// TwinCAT 3 PLC project mover_demo
// ProgramVersion: 3.1.4024.12
// libraries:
//   CmpBitmapPool, * (System)
//   Tc2_Math, * (Beckhoff Automation GmbH)
//   Tc2_MC2, * (Beckhoff Automation GmbH)
//   Tc2_MC2_Drive, * (Beckhoff Automation GmbH)
//   Tc2_Standard, * (Beckhoff Automation GmbH)
//   Tc2_System, * (Beckhoff Automation GmbH)
//   Tc2_Utilities, * (Beckhoff Automation GmbH)
//   Tc3_JsonXml, * (Beckhoff Automation GmbH)
//   Tc3_Module, * (Beckhoff Automation GmbH)
//   VisuDialogs, * (System)
//   VisuSymbols,3.5.10.0,System
// project tree:
//   DUTs/Helptec/Axis/ AxisBase_t.TcDUT, AxisBeckhoff_t.TcDUT, AxisLinMotConst_t.TcDUT (not stored), AxisLinMot_t.TcDUT, AxisSMC_t.TcDUT (not stored), typeInputArea.TcDUT, typeOutputArea.TcDUT
//   DUTs/Helptec/ Cylinder2Pos_config.TcDUT, enLamp.TcDUT (not stored), enState.TcDUT (not stored), structAlarm.TcDUT (not stored), structButton.TcDUT
//   DUTs/Helptec/Recipe/ RecipeAxisLinear2Pos_t.TcDUT
//   DUTs/Helptec/RS_Axis/ FeederDelays_t.TcDUT (not stored), MoveProfile1D_t.TcDUT, MoveProfile_t.TcDUT, TriggerType_e.TcDUT, VectorMove1D_t.TcDUT
//   DUTs/ PieceType_e.TcTLEO (not stored), Mover_st.TcDUT (not stored), Piece_st.TcDUT (not stored)
//   / GlobalTextList.TcGTLO (excluded from build), PlcTask.TcTTO, Visualization Manager.TcVMO (not stored), VISU_TASK.TcTTO
//   GVLs/ AXIS.TcGVL, CONST.TcGVL, GVL.TcGVL, HMI.TcGVL, IN.TcGVL, IO_BOX.TcGVL, OUT.TcGVL, PERS.TcGVL, SIMU.TcGVL
//   POUs/00_MAIN/FB%27s/ FB_Safety.TcPOU (not stored)
//   POUs/00_MAIN/ MAIN.TcPOU, _02_SAFETY.TcPOU, _05_FLAGS.TcPOU (not stored)
//   POUs/10_HMI/FB%27s/ FB_BUTTON.TcPOU (not stored), FB_HMI_BT.TcPOU (not stored), FB_Keba_key.TcPOU (not stored), FB_LampeBNI007F.TcPOU (not stored), FB_STATE.TcPOU (not stored)
//   POUs/10_HMI/ _10_HMI.TcPOU, _11_PAR_CHK.TcPOU (not stored), _14_STATE.TcPOU
//   POUs/20_AUTO/ Axis_e.TcTLEO, LinearAxis_e.TcTLEO, RecipeType_e.TcTLEO, Recipe_21_101_t.TcDUT, StationList_e.TcTLEO, _20_AUTO.TcPOU, _21_CopyDefaultRecipe.TcPOU
//   POUs/20_AUTO/BuR SuperTrack com/ CT_Shuttle_BR_to_Tc_Status_t.TcDUT, CT_Shuttle_BR_to_Tc_t.TcDUT, CT_Shuttle_BR_to_Tc_u.TcDUT, CT_Shuttle_Tc_To_BR_Command_t.TcDUT, CT_Shuttle_Tc_to_BR_t.TcDUT, CT_Shuttle_Tc_to_BR_u.TcDUT, CT_Track_BR_to_TC_Status_t.TcDUT, CT_Track_BR_to_Tc_t.TcDUT, CT_Track_BR_to_Tc_u.TcDUT, CT_Track_Tc_to_BR_Command_t.TcDUT, CT_Track_Tc_to_BR_t.TcDUT, CT_Track_Tc_to_BR_u.TcDUT, gMoverAxis.TcGVL
//   POUs/20_AUTO/FB%27s/Alarm/ FB_ALARM.TcPOU (not stored), FB_ALARM32.TcPOU (not stored)
//   POUs/20_AUTO/FB%27s/ FB_WandlerForceSensor.TcPOU (not stored), getPercent.TcPOU (not stored)
//   POUs/20_AUTO/FB%27s/RS Axis/ BowlBandFeeder_Config_t.TcDUT (not stored), FB_AUT_Statistics.TcPOU (not stored), FB_BowlBandFeeder.TcPOU (not stored), FB_Feeder2Sensors.TcPOU (not stored), FB_Fifo.TcPOU (not stored), FB_LinearMotionMan.TcPOU (not stored), LinearMotionMan_Config_t.TcDUT (not stored)
//   POUs/20_AUTO/FB%27s/Achsen/ FB_AxisLIN_V1_1.TcPOU (not stored), FB_AxisLMturn_V1_1.TcPOU (not stored), FB_AxisLM_V1_1.TcPOU (not stored), FB_AxisRotTable_V1_1.TcPOU (not stored), FB_AxisSMC_V1_1.TcPOU (not stored), FB_AxisTURN_V1_1.TcPOU (not stored), JXCE1_Baustein.TcPOU (not stored)
//   POUs/20_AUTO/FB%27s/Pneumatic/ FB_ZylMo2El_V2_1.TcPOU (not stored)
//   POUs/20_AUTO/FB%27s/Vorlagen/ FB_ABL_VORLAGE.TcPOU (not stored), POU_AUT_VORLAGE.TcPOU (not stored), POU_ERR_VORLAGE.TcPOU (not stored), _01_MAIN.TcPOU (not stored)
//   POUs/20_AUTO/FileMan/ FB_FileMan.TcPOU, FileMan.TcPOU, LoadFromMemory.TcPOU, ReadJsonDom.TcPOU, SaveInMemory.TcPOU, SaveInMemory_Recipe.TcPOU
//   POUs/20_AUTO/Mover/ ApproachScenario_e.TcTLEO, DistToTravel.TcPOU, FB_Group.TcPOU, FB_Mover.TcPOU, FB_MoverMan.TcPOU, FB_Position.TcPOU, FB_SimuMoverAxis.TcPOU, FB_Station.TcPOU, FB_PieceHolder.TcPOU, FB_StationMan.TcPOU, IProcessSampleMover.TcIO (not stored), ISimuMoverTimers.TcIO, IStation.TcIO, MoverDirection_e.TcTLEO, MoverState_e.TcTLEO, VISU_MoverDetail.TcVIS, VISU_MoverView.TcVIS, Pos2D_t.TcDUT (not stored), ProcessExec_e.TcDUT (not stored), StationName_e.TcTLEO
//   POUs/20_AUTO/Simu/ FB_Simu_AxisLIN_V1_1.TcPOU, FB_Simu_AxisLM_V1_1.TcPOU, FB_Simu_Feeder.TcPOU, FB_Simu_Zyl2Pos.TcPOU
//   POUs/20_AUTO/ST100/ FB_ABL_LASER.TcPOU, FB_AUT_LASER.TcPOU, FB_AUT_100.TcPOU, F_GetPercent.TcPOU (not stored), F_GetPercent_2.TcPOU, ST100_Load_e.TcTLEO (not stored), FB_ABL_LOAD.TcPOU, FB_ABL_MODIFY.TcPOU, FB_ABL_UNLOAD.TcPOU, FB_AUT_ABSTRACT.TcPOU, FB_ABL_100.TcPOU (not stored), FB_AUT_LOAD.TcPOU, FB_AUT_MODIFY.TcPOU, FB_AUT_UNLOAD.TcPOU, ProcessExecution_e.TcTLEO (not stored), ST100_e.TcTLEO (not stored), ST100_Modify_e.TcTLEO (not stored), ST100_Laser_e.TcTLEO, ST100_Unload_e.TcTLEO (not stored)
//   POUs/20_AUTO/ST105/Fanuc_robot/ Fanuc_command_ext_to_robot_t.TcDUT (not stored), Fanuc_command_std_to_robot_t.TcDUT, Fanuc_hw_command_to_robot_t.TcDUT (not stored), Fanuc_status_std_from_robot.TcDUT (not stored), ST105_Fanuc_command_t.TcDUT, ST105_Fanuc_status_t.TcDUT
//   POUs/20_AUTO/ST105/ FB_ABL_105_Feeder.TcPOU, FB_ABL_105_Pnp.TcPOU, FB_AUT_105.TcPOU, ST105_Axis.TcGVL, ST105_PnpVerPushPos_e.TcDUT, ST105_Recipe_t.TcDUT, ST105_Feeder_e.TcDUT, ST105_Pnp_e.TcTLEO, ST105_Slider_e.TcDUT, ST105_Cylinders_e.TcTLEO, VISU_Recipe_ST105.TcVIS, VISU_ST105.TcVIS
//   POUs/20_AUTO/ST110/ POU_ALARM_110.TcPOU, ST110_Alarm_e.TcDUT, ST110_Cylinders_e.TcTLEO (not stored), ST110_Feeder_e.TcDUT, FB_ABL_110_Feeder.TcPOU, FB_ABL_110_Pnp.TcPOU, FB_AUT_110.TcPOU, ST110_Axis.TcGVL, ST110_PnpVerPushPos_e.TcDUT, ST110_Pnp_e.TcTLEO, ST110_PnpHorPos_e.TcDUT, ST110_PnpVerPos_e.TcDUT, ST110_Recipe_t.TcDUT, VISU_Recipe_ST110.TcVIS, VISU_ST110.TcVIS
//   POUs/20_AUTO/ST115/ FB_ABL_115_Feeder.TcPOU, FB_ABL_115_Pnp.TcPOU, FB_AUT_115.TcPOU, ST115_PnpVerPushPos_e.TcDUT, ST115_Cylinders_e.TcTLEO, ST115_Recipe_t.TcDUT, ST115_Axis.TcGVL, ST115_Feeder_e.TcDUT, ST115_PnpHorPos_e.TcDUT, ST115_PnpVerPos_e.TcDUT (not stored), ST115_Pnp_e.TcTLEO, VISU_Recipe_ST115.TcVIS, VISU_ST115.TcVIS
//   POUs/20_AUTO/ST120/ FB_ABL_120_Feeder.TcPOU, FB_ABL_120_Pnp.TcPOU, FB_AUT_120.TcPOU, POU_ALARM_120.TcPOU (not stored), ST120_Alarm_e.TcDUT (not stored), ST120_Cylinders_e.TcTLEO, ST120_Axis.TcGVL, ST120_Feeder_e.TcDUT, ST120_PnpHorPos_e.TcDUT (not stored), ST120_PnpVerPos_e.TcDUT, ST120_Pnp_e.TcTLEO, ST120_Recipe_t.TcDUT, VISU_Recipe_ST120.TcVIS, VISU_ST120.TcVIS
//   POUs/20_AUTO/ST125/ FB_ABL_125_Feeder.TcPOU, FB_ABL_125_Pnp.TcPOU, FB_AUT_125.TcPOU, POU_ALARM_125.TcPOU, ST125_Alarm_e.TcDUT, ST125_Cylinders_e.TcTLEO, ST125_Axis.TcGVL, ST125_Feeder_e.TcDUT, ST125_PnpHorPos_e.TcDUT, ST125_PnpVerPos_e.TcDUT, ST125_Pnp_e.TcTLEO, ST125_Recipe_t.TcDUT, VISU_Recipe_ST125.TcVIS, VISU_ST125.TcVIS
//   POUs/20_AUTO/ST128/ FB_ABL_128_TubeCapCheck.TcPOU, FB_AUT_128.TcPOU, ST128_TubeCapCheck_e.TcTLEO (not stored), ST128_Recipe_t.TcDUT, VISU_Recipe_ST128.TcVIS (not stored), VISU_ST128.TcVIS
//   POUs/20_AUTO/ST130/ FB_ABL_130_Dose.TcPOU, FB_ABL_MODIFY_135.TcPOU, FB_AUT_130.TcPOU, FB_AUT_135.TcPOU, ST130_Axis.TcGVL, ST130_Cylinders_e.TcTLEO, ST130_DosierkammerPos_e.TcDUT (not stored), ST130_PatroneAushebenPos_e.TcDUT, ST130_Recipe_t.TcDUT, ST130_Dose_e.TcTLEO, VISU_Recipe_ST130.TcVIS, VISU_ST130.TcVIS
//   POUs/20_AUTO/ST140/ FB_ABL_140_Measure.TcPOU, FB_AUT_140.TcPOU, LaserPlace_e.TcDUT, ST140_Measure_e.TcTLEO, ST140_Recipe_t.TcDUT, VISU_Recipe_ST140.TcVIS, VISU_ST140.TcVIS
//   POUs/20_AUTO/ST145/ FB_ABL_145_Feeder.TcPOU, FB_ABL_145_Pnp.TcPOU, FB_AUT_145.TcPOU, ST145_Axis.TcGVL, ST145_Cylinders_e.TcTLEO (not stored), ST145_Feeder_e.TcDUT, ST145_PnpHorPos_e.TcDUT, ST145_PnpVerPos_e.TcDUT, ST145_Recipe_t.TcDUT, ST145_Pnp_e.TcTLEO, VISU_Recipe_ST145.TcVIS, VISU_ST145.TcVIS
//   POUs/20_AUTO/ST15x/ FB_ABL_150.TcPOU, FB_ABL_150_solo.TcPOU, FB_AUT_150.TcPOU, FB_AUT_155.TcPOU, ST150_Cylinders_e.TcTLEO, ST150_Uss_e.TcTLEO, ST150_Recipe_t.TcDUT (not stored), Ultrasonic_IN_bits_t.TcDUT, Ultrasonic_OUT_bits_t.TcDUT, VISU_Recipe_ST150.TcVIS, VISU_ST150.TcVIS
//   POUs/20_AUTO/ST16x/CETA/ CETA_error_handling_t.TcDUT, CETA_IN_bits_t.TcDUT, CETA_IN_u.TcDUT, CETA_IO.TcGVL, CETA_OUT_bits_t.TcDUT, CETA_OUT_u.TcDUT, CETA_Result_e.TcDUT, CETA_Unit_e.TcDUT, FB_CETA_715.TcPOU
//   POUs/20_AUTO/ST16x/CETA/CETA_Measurement_t/ CETA_Measurement_block1_t.TcDUT (not stored), CETA_Measurement_block2_t.TcDUT, CETA_Measurement_block3_t.TcDUT (not stored), CETA_Measurement_t.TcDUT, CETA_Res_Data_t.TcDUT
//   POUs/20_AUTO/ST16x/CETA/CETA_Parameter_blocks/ CETA_Parameter_blocks_t.TcDUT
//   POUs/20_AUTO/ST16x/CETA/CETA_com_union/ CETA_Parameter_blocks_u.TcDUT
//   POUs/20_AUTO/ST16x/ FB_ABL_160.TcPOU, FB_AUT_160.TcPOU, FB_AUT_165.TcPOU, ST160_PnpVerPos_e.TcDUT, ST16x_Axis.TcGVL, ST160_Cylinders_e.TcTLEO, ST160_Recipe_t.TcDUT, ST160_CETA_e.TcTLEO, VISU_Recipe_ST160.TcVIS, VISU_ST160.TcVIS
//   POUs/20_AUTO/ST170/ FB_ABL_170.TcPOU, FB_AUT_170.TcPOU, ST170_Axis.TcGVL (not stored), ST170_RFID_e.TcTLEO, ST170_PnpVerPos_e.TcDUT, ST170_Recipe_t.TcDUT, VISU_Recipe_ST170.TcVIS, VISU_ST170.TcVIS
//   POUs/20_AUTO/ST175/ FB_ABL_175.TcPOU, FB_AUT_175.TcPOU, ST175_LASER_e.TcTLEO, ST175_Cylinders_e.TcTLEO, ST175_Recipe_t.TcDUT, VISU_Recipe_ST175.TcVIS, VISU_ST175.TcVIS (not stored)
//   POUs/20_AUTO/ST175/Trumpf/ FB_Laser_ABL.TcPOU, if_BitCommand_u.TcDUT (not stored), if_Command_t.TcDUT, if_Command_u.TcDUT, if_SingleCmds.TcGVL (not stored), if_TruMark.TcGVL, TruMarkLaserStatus.TcDUT (not stored), TruMark_Ethercat_dj.TcPOU, TruMark_SingleCmds.TcPOU
//   POUs/20_AUTO/ST180/ FB_ABL_180_Pnp.TcPOU, FB_AUT_180.TcPOU, ST180_Axis.TcGVL, ST180_Cylinders_e.TcTLEO, ST180_PnpHorPos_e.TcDUT (not stored), ST180_PnpVerPos_e.TcDUT, ST180_Pnp_e.TcTLEO, ST180_Recipe_t.TcDUT, VISU_Recipe_ST180.TcVIS, VISU_ST180.TcVIS
//   POUs/20_AUTO/ST185/ FB_ABL_185_Pnp.TcPOU, FB_AUT_185.TcPOU, ST185_Axis.TcGVL, ST185_Cylinders_e.TcTLEO, ST185_PnpHorPos_e.TcDUT, ST185_PnpVerPos_e.TcDUT, ST185_Pnp_e.TcTLEO, ST185_Recipe_t.TcDUT, VISU_Recipe_ST185.TcVIS, VISU_ST185.TcVIS (not stored)
//   POUs/20_AUTO/TOOL/ ASSERT.TcPOU, EqualApproximately.TcPOU (not stored), EqualDelta.TcPOU (not stored), EqualEssentially.TcPOU (not stored), GetTick.TcPOU, IObject.TcIO, MAP_REAL_TO_INT.TcPOU, SortBubbleLREAL.TcPOU (not stored)
//   VISUs/ Custom.TcIPO (not stored), VISU_LinearConfigArray.TcVIS, VISU_Cylinder2PosConfig.TcVIS, VISU_AxisManual.TcVIS, VISU_main.TcVIS, VISU_Time.TcVIS
// real-time tasks:
//   TASK PlcTask: cycle T#10ms, priority 20, ADS port 350
//   TASK VISU_TASK: cycle T#10ms, priority 21, ADS port 351
//   TASK Task_fileMan: cycle T#100000us, priority 45, ADS port 352
// motion (NC):
//   TASK NC-Task 1 SAF: cycle T#2ms, priority 4, ADS port 501
//   TASK NC-Task 1 SVB: cycle T#10ms, priority 8, ADS port 511
//   AXIS ST110_01Y (id 1)
//     Dynamic: AccelerationMaximum=100000, DecelerationMaximum=100000, Acceleration=40000, Deceleration=40000, Jerk=800000
//     OtherSettings: AllowMotionCmdToSlave=true
//     encoder EncType=1
//       SoftEndMinControl: Enable=true, Range=-5
//     drive DrvType=5
//       Analog: TorqueSetpointScale=10, ScaleFactorActTorque=0.1
//       TimeComp: TaskDelayCycles=1
//     controller CtrType=1
//       CtrPara: PriorControlFactor=1
//         Observer: BandWidth=20
//   AXIS ST110_02Z (id 2)
//     Dynamic: AccelerationMaximum=100000, DecelerationMaximum=100000, Acceleration=15000, Deceleration=15000, Jerk=10000000
//     OtherSettings: AllowMotionCmdToSlave=true
//     encoder EncType=1
//       SoftEndMinControl: Enable=true, Range=-5
//     drive DrvType=5
//       Analog: TorqueSetpointScale=10, ScaleFactorActTorque=0.1
//       TimeComp: TaskDelayCycles=1
//     controller CtrType=1
//       CtrPara: PriorControlFactor=1
//         Observer: BandWidth=20
//   AXIS ST110_03Z (id 3)
//     Dynamic: AccelerationMaximum=100000, DecelerationMaximum=100000, Acceleration=15000, Deceleration=15000, Jerk=10000000
//     OtherSettings: AllowMotionCmdToSlave=true
//     encoder EncType=1
//       SoftEndMinControl: Enable=true, Range=-5
//     drive DrvType=5
//       Analog: TorqueSetpointScale=10, ScaleFactorActTorque=0.1
//       TimeComp: TaskDelayCycles=1
//     controller CtrType=1
//       CtrPara: PriorControlFactor=1
//         Observer: BandWidth=20
//   AXIS ST110_04Z (id 11)
//     OtherSettings: AllowMotionCmdToSlave=true
//     encoder EncType=1
//     drive DrvType=5
//       Analog: TorqueSetpointScale=10, ScaleFactorActTorque=0.1
//       TimeComp: TaskDelayCycles=1
//     controller CtrType=1
//       CtrPara: PriorControlFactor=1
//         Observer: BandWidth=20
//   AXIS ST110_10W (id 4)
//     General: UnitName=°, UnitFlags=#x00000004
//     Dynamic: AccelerationMaximum=36000, DecelerationMaximum=36000, Acceleration=3600, Deceleration=3600, Jerk=3600000
//     Velo: Maximum=360
//     OtherSettings: AllowMotionCmdToSlave=true
//     encoder EncType=1
//     drive DrvType=5
//       Analog: VeloReferenz=360, TorqueSetpointScale=10, ScaleFactorActTorque=0.1
//       TimeComp: TaskDelayCycles=1
//     controller CtrType=1
//       CtrPara: PriorControlFactor=1
//         Observer: BandWidth=20
//   AXIS ST115_01Y (id 5)
//     OtherSettings: AllowMotionCmdToSlave=true
//     encoder EncType=1
//     drive DrvType=5
//       Analog: TorqueSetpointScale=10, ScaleFactorActTorque=0.1
//       TimeComp: TaskDelayCycles=1
//     controller CtrType=1
//       CtrPara: PriorControlFactor=1
//         Observer: BandWidth=20
//   AXIS ST115_02Z (id 6)
//     OtherSettings: AllowMotionCmdToSlave=true
//     encoder EncType=1
//     drive DrvType=5
//       Analog: TorqueSetpointScale=10, ScaleFactorActTorque=0.1
//       TimeComp: TaskDelayCycles=1
//     controller CtrType=1
//       CtrPara: PriorControlFactor=1
//         Observer: BandWidth=20
//   AXIS ST115_03Z (id 7)
//     OtherSettings: AllowMotionCmdToSlave=true
//     encoder EncType=1
//     drive DrvType=5
//       Analog: TorqueSetpointScale=10, ScaleFactorActTorque=0.1
//       TimeComp: TaskDelayCycles=1
//     controller CtrType=1
//       CtrPara: PriorControlFactor=1
//         Observer: BandWidth=20
//   AXIS ST115_04Z (id 12)
//     OtherSettings: AllowMotionCmdToSlave=true
//     encoder EncType=1
//     drive DrvType=5
//       Analog: TorqueSetpointScale=10, ScaleFactorActTorque=0.1
//       TimeComp: TaskDelayCycles=1
//     controller CtrType=1
//       CtrPara: PriorControlFactor=1
//         Observer: BandWidth=20
//   AXIS ST115_10W (id 8)
//     General: UnitName=°
//     OtherSettings: AllowMotionCmdToSlave=true
//     encoder EncType=1
//     drive DrvType=5
//       Analog: TorqueSetpointScale=10, ScaleFactorActTorque=0.1
//       TimeComp: TaskDelayCycles=1
//     controller CtrType=1
//       CtrPara: PriorControlFactor=1
//         Observer: BandWidth=20
//   AXIS ST120_01Y (id 9)
//     OtherSettings: AllowMotionCmdToSlave=true
//     encoder EncType=1
//     drive DrvType=5
//       Analog: TorqueSetpointScale=10, ScaleFactorActTorque=0.1
//       TimeComp: TaskDelayCycles=1
//     controller CtrType=1
//       CtrPara: PriorControlFactor=1
//         Observer: BandWidth=20
//   AXIS ST120_02Z (id 10)
//     OtherSettings: AllowMotionCmdToSlave=true
//     encoder EncType=1
//     drive DrvType=5
//       Analog: TorqueSetpointScale=10, ScaleFactorActTorque=0.1
//       TimeComp: TaskDelayCycles=1
//     controller CtrType=1
//       CtrPara: PriorControlFactor=1
//         Observer: BandWidth=20
//   AXIS ST125_01Y (id 13)
//     OtherSettings: AllowMotionCmdToSlave=true
//     encoder EncType=1
//     drive DrvType=5
//       Analog: TorqueSetpointScale=10, ScaleFactorActTorque=0.1
//       TimeComp: TaskDelayCycles=1
//     controller CtrType=1
//       CtrPara: PriorControlFactor=1
//         Observer: BandWidth=20
//   AXIS ST125_02Z (id 14)
//     OtherSettings: AllowMotionCmdToSlave=true
//     encoder EncType=1
//     drive DrvType=5
//       Analog: TorqueSetpointScale=10, ScaleFactorActTorque=0.1
//       TimeComp: TaskDelayCycles=1
//     controller CtrType=1
//       CtrPara: PriorControlFactor=1
//         Observer: BandWidth=20
//   AXIS ST125_10W (id 15)
//     General: UnitName=°
//     OtherSettings: AllowMotionCmdToSlave=true
//     encoder EncType=1
//     drive DrvType=5
//       Analog: TorqueSetpointScale=10, ScaleFactorActTorque=0.1
//       TimeComp: TaskDelayCycles=1
//     controller CtrType=1
//       CtrPara: PriorControlFactor=1
//         Observer: BandWidth=20
//   AXIS SIMU_ST145_01Y (id 16)
//     OtherSettings: AllowMotionCmdToSlave=true
//     encoder EncType=1
//     drive DrvType=5
//       Analog: TorqueSetpointScale=10, ScaleFactorActTorque=0.1
//       TimeComp: TaskDelayCycles=1
//     controller CtrType=1
//       CtrPara: PriorControlFactor=1
//         Observer: BandWidth=20
//   AXIS SIMU_ST145_02Z (id 17)
//     OtherSettings: AllowMotionCmdToSlave=true
//     encoder EncType=1
//     drive DrvType=5
//       Analog: TorqueSetpointScale=10, ScaleFactorActTorque=0.1
//       TimeComp: TaskDelayCycles=1
//     controller CtrType=1
//       CtrPara: PriorControlFactor=1
//         Observer: BandWidth=20
//   AXIS ST145_10W (id 18)
//     General: UnitName=°
//     OtherSettings: AllowMotionCmdToSlave=true
//     encoder EncType=1
//     drive DrvType=5
//       Analog: TorqueSetpointScale=10, ScaleFactorActTorque=0.1
//       TimeComp: TaskDelayCycles=1
//     controller CtrType=1
//       CtrPara: PriorControlFactor=1
//         Observer: BandWidth=20
//   AXIS ST160_01Z (id 27)
//     OtherSettings: AllowMotionCmdToSlave=true
//     encoder EncType=1
//     drive DrvType=5
//       Analog: TorqueSetpointScale=10, ScaleFactorActTorque=0.1
//       TimeComp: TaskDelayCycles=1
//     controller CtrType=1
//       CtrPara: PriorControlFactor=1
//         Observer: BandWidth=20
//   AXIS ST165_01Z (id 28)
//     OtherSettings: AllowMotionCmdToSlave=true
//     encoder EncType=1
//     drive DrvType=5
//       Analog: TorqueSetpointScale=10, ScaleFactorActTorque=0.1
//       TimeComp: TaskDelayCycles=1
//     controller CtrType=1
//       CtrPara: PriorControlFactor=1
//         Observer: BandWidth=20
//   AXIS ST170_01Z (id 19)
//     OtherSettings: AllowMotionCmdToSlave=true
//     encoder EncType=1
//     drive DrvType=5
//       Analog: TorqueSetpointScale=10, ScaleFactorActTorque=0.1
//       TimeComp: TaskDelayCycles=1
//     controller CtrType=1
//       CtrPara: PriorControlFactor=1
//         Observer: BandWidth=20
//   AXIS ST180_01Y (id 20)
//     OtherSettings: AllowMotionCmdToSlave=true
//     encoder EncType=1
//     drive DrvType=5
//       Analog: TorqueSetpointScale=10, ScaleFactorActTorque=0.1
//       TimeComp: TaskDelayCycles=1
//     controller CtrType=1
//       CtrPara: PriorControlFactor=1
//         Observer: BandWidth=20
//   AXIS ST180_02Z (id 21)
//     OtherSettings: AllowMotionCmdToSlave=true
//     encoder EncType=1
//     drive DrvType=5
//       Analog: TorqueSetpointScale=10, ScaleFactorActTorque=0.1
//       TimeComp: TaskDelayCycles=1
//     controller CtrType=1
//       CtrPara: PriorControlFactor=1
//         Observer: BandWidth=20
//   AXIS ST180_10Z (id 22)
//     OtherSettings: AllowMotionCmdToSlave=true
//     encoder EncType=1
//     drive DrvType=5
//       Analog: TorqueSetpointScale=10, ScaleFactorActTorque=0.1
//       TimeComp: TaskDelayCycles=1
//     controller CtrType=1
//       CtrPara: PriorControlFactor=1
//         Observer: BandWidth=20
//   AXIS ST185_01Y (id 23)
//     OtherSettings: AllowMotionCmdToSlave=true
//     encoder EncType=1
//     drive DrvType=5
//       Analog: TorqueSetpointScale=10, ScaleFactorActTorque=0.1
//       TimeComp: TaskDelayCycles=1
//     controller CtrType=1
//       CtrPara: PriorControlFactor=1
//         Observer: BandWidth=20
//   AXIS ST185_02Z (id 24)
//     OtherSettings: AllowMotionCmdToSlave=true
//     encoder EncType=1
//     drive DrvType=5
//       Analog: TorqueSetpointScale=10, ScaleFactorActTorque=0.1
//       TimeComp: TaskDelayCycles=1
//     controller CtrType=1
//       CtrPara: PriorControlFactor=1
//         Observer: BandWidth=20
//   AXIS ST185_10Z (id 25)
//     OtherSettings: AllowMotionCmdToSlave=true
//     encoder EncType=1
//     drive DrvType=5
//       Analog: TorqueSetpointScale=10, ScaleFactorActTorque=0.1
//       TimeComp: TaskDelayCycles=1
//     controller CtrType=1
//       CtrPara: PriorControlFactor=1
//         Observer: BandWidth=20
//   AXIS Axis 34 (id 34)
//     OtherSettings: AllowMotionCmdToSlave=true
//     encoder EncType=19
//       EncPara: MaxCount=#xffffffff
//     drive DrvType=16
//       DrvPara: MaxCount=#xffffffff
//         Analog: TorqueSetpointScale=10, ScaleFactorActTorque=0.1
//         TimeComp: TaskDelayCycles=1
//     controller CtrType=1
//       CtrPara: PriorControlFactor=1
//         Observer: BandWidth=20
//   AXIS Axis 35 (id 35)
//     OtherSettings: AllowMotionCmdToSlave=true
//     encoder EncType=19
//       EncPara: MaxCount=#xffffffff
//     drive DrvType=16
//       DrvPara: MaxCount=#xffffffff
//         Analog: TorqueSetpointScale=10, ScaleFactorActTorque=0.1
//         TimeComp: TaskDelayCycles=1
//     controller CtrType=1
//       CtrPara: PriorControlFactor=1
//         Observer: BandWidth=20
//   AXIS Axis 36 (id 36)
//     OtherSettings: AllowMotionCmdToSlave=true
//     encoder EncType=19
//       EncPara: MaxCount=#xffffffff
//     drive DrvType=16
//       DrvPara: MaxCount=#xffffffff
//         Analog: TorqueSetpointScale=10, ScaleFactorActTorque=0.1
//         TimeComp: TaskDelayCycles=1
//     controller CtrType=1
//       CtrPara: PriorControlFactor=1
//         Observer: BandWidth=20
//   AXIS Axis 37 (id 37)
//     OtherSettings: AllowMotionCmdToSlave=true
//     encoder EncType=19
//       EncPara: MaxCount=#xffffffff
//     drive DrvType=16
//       DrvPara: MaxCount=#xffffffff
//         Analog: TorqueSetpointScale=10, ScaleFactorActTorque=0.1
//         TimeComp: TaskDelayCycles=1
//     controller CtrType=1
//       CtrPara: PriorControlFactor=1
//         Observer: BandWidth=20
//   AXIS Axis 38 (id 38)
//     OtherSettings: AllowMotionCmdToSlave=true
//     encoder EncType=19
//       EncPara: MaxCount=#xffffffff
//     drive DrvType=16
//       DrvPara: MaxCount=#xffffffff
//         Analog: TorqueSetpointScale=10, ScaleFactorActTorque=0.1
//         TimeComp: TaskDelayCycles=1
//     controller CtrType=1
//       CtrPara: PriorControlFactor=1
//         Observer: BandWidth=20
//   AXIS Axis 39 (id 39)
//     OtherSettings: AllowMotionCmdToSlave=true
//     encoder EncType=19
//       EncPara: MaxCount=#xffffffff
//     drive DrvType=16
//       DrvPara: MaxCount=#xffffffff
//         Analog: TorqueSetpointScale=10, ScaleFactorActTorque=0.1
//         TimeComp: TaskDelayCycles=1
//     controller CtrType=1
//       CtrPara: PriorControlFactor=1
//         Observer: BandWidth=20
//   AXIS Axis 40 (id 40)
//     OtherSettings: AllowMotionCmdToSlave=true
//     encoder EncType=19
//       EncPara: MaxCount=#xffffffff
//     drive DrvType=16
//       DrvPara: MaxCount=#xffffffff
//         Analog: TorqueSetpointScale=10, ScaleFactorActTorque=0.1
//         TimeComp: TaskDelayCycles=1
//     controller CtrType=1
//       CtrPara: PriorControlFactor=1
//         Observer: BandWidth=20
//   AXIS Axis 41 (id 41)
//     OtherSettings: AllowMotionCmdToSlave=true
//     encoder EncType=19
//       EncPara: MaxCount=#xffffffff
//     drive DrvType=16
//       DrvPara: MaxCount=#xffffffff
//         Analog: TorqueSetpointScale=10, ScaleFactorActTorque=0.1
//         TimeComp: TaskDelayCycles=1
//     controller CtrType=1
//       CtrPara: PriorControlFactor=1
//         Observer: BandWidth=20
//   AXIS Axis 42 (id 42)
//     OtherSettings: AllowMotionCmdToSlave=true
//     encoder EncType=19
//       EncPara: MaxCount=#xffffffff
//     drive DrvType=16
//       DrvPara: MaxCount=#xffffffff
//         Analog: TorqueSetpointScale=10, ScaleFactorActTorque=0.1
//         TimeComp: TaskDelayCycles=1
//     controller CtrType=1
//       CtrPara: PriorControlFactor=1
//         Observer: BandWidth=20
//   AXIS Axis 43 (id 43)
//     OtherSettings: AllowMotionCmdToSlave=true
//     encoder EncType=19
//       EncPara: MaxCount=#xffffffff
//     drive DrvType=16
//       DrvPara: MaxCount=#xffffffff
//         Analog: TorqueSetpointScale=10, ScaleFactorActTorque=0.1
//         TimeComp: TaskDelayCycles=1
//     controller CtrType=1
//       CtrPara: PriorControlFactor=1
//         Observer: BandWidth=20
//   AXIS Axis 44 (id 44)
//     OtherSettings: AllowMotionCmdToSlave=true
//     encoder EncType=19
//       EncPara: MaxCount=#xffffffff
//     drive DrvType=16
//       DrvPara: MaxCount=#xffffffff
//         Analog: TorqueSetpointScale=10, ScaleFactorActTorque=0.1
//         TimeComp: TaskDelayCycles=1
//     controller CtrType=1
//       CtrPara: PriorControlFactor=1
//         Observer: BandWidth=20
//   AXIS Axis 45 (id 45)
//     OtherSettings: AllowMotionCmdToSlave=true
//     encoder EncType=19
//       EncPara: MaxCount=#xffffffff
//     drive DrvType=16
//       DrvPara: MaxCount=#xffffffff
//         Analog: TorqueSetpointScale=10, ScaleFactorActTorque=0.1
//         TimeComp: TaskDelayCycles=1
//     controller CtrType=1
//       CtrPara: PriorControlFactor=1
//         Observer: BandWidth=20
//   AXIS Axis 46 (id 46)
//     OtherSettings: AllowMotionCmdToSlave=true
//     encoder EncType=19
//       EncPara: MaxCount=#xffffffff
//     drive DrvType=16
//       DrvPara: MaxCount=#xffffffff
//         Analog: TorqueSetpointScale=10, ScaleFactorActTorque=0.1
//         TimeComp: TaskDelayCycles=1
//     controller CtrType=1
//       CtrPara: PriorControlFactor=1
//         Observer: BandWidth=20
//   AXIS Axis 47 (id 47)
//     OtherSettings: AllowMotionCmdToSlave=true
//     encoder EncType=19
//       EncPara: MaxCount=#xffffffff
//     drive DrvType=16
//       DrvPara: MaxCount=#xffffffff
//         Analog: TorqueSetpointScale=10, ScaleFactorActTorque=0.1
//         TimeComp: TaskDelayCycles=1
//     controller CtrType=1
//       CtrPara: PriorControlFactor=1
//         Observer: BandWidth=20
//   AXIS Axis 48 (id 48)
//     OtherSettings: AllowMotionCmdToSlave=true
//     encoder EncType=19
//       EncPara: MaxCount=#xffffffff
//     drive DrvType=16
//       DrvPara: MaxCount=#xffffffff
//         Analog: TorqueSetpointScale=10, ScaleFactorActTorque=0.1
//         TimeComp: TaskDelayCycles=1
//     controller CtrType=1
//       CtrPara: PriorControlFactor=1
//         Observer: BandWidth=20
//   AXIS Axis 49 (id 49)
//     OtherSettings: AllowMotionCmdToSlave=true
//     encoder EncType=19
//       EncPara: MaxCount=#xffffffff
//     drive DrvType=16
//       DrvPara: MaxCount=#xffffffff
//         Analog: TorqueSetpointScale=10, ScaleFactorActTorque=0.1
//         TimeComp: TaskDelayCycles=1
//     controller CtrType=1
//       CtrPara: PriorControlFactor=1
//         Observer: BandWidth=20
//   AXIS Axis 50 (id 50)
//     OtherSettings: AllowMotionCmdToSlave=true
//     encoder EncType=19
//       EncPara: MaxCount=#xffffffff
//     drive DrvType=16
//       DrvPara: MaxCount=#xffffffff
//         Analog: TorqueSetpointScale=10, ScaleFactorActTorque=0.1
//         TimeComp: TaskDelayCycles=1
//     controller CtrType=1
//       CtrPara: PriorControlFactor=1
//         Observer: BandWidth=20
//   AXIS ST145_01Y (id 51)
//     OtherSettings: AllowMotionCmdToSlave=true
//     encoder EncType=19
//       EncPara: MaxCount=#xffffffff
//     drive DrvType=16
//       DrvPara: MaxCount=#xffffffff
//         Analog: TorqueSetpointScale=10, ScaleFactorActTorque=0.1
//         TimeComp: TaskDelayCycles=1
//     controller CtrType=1
//       CtrPara: PriorControlFactor=1
//         PosDiffControl: Enable=false
//         Observer: BandWidth=20
//   AXIS ST145_02Z (id 52)
//     OtherSettings: AllowMotionCmdToSlave=true
//     encoder EncType=19
//       EncPara: MaxCount=#xffffffff
//     drive DrvType=16
//       DrvPara: MaxCount=#xffffffff
//         Analog: TorqueSetpointScale=10, ScaleFactorActTorque=0.1
//         TimeComp: TaskDelayCycles=1
//     controller CtrType=1
//       CtrPara: PriorControlFactor=1
//         PosDiffControl: Enable=false
//         Observer: BandWidth=20
//   AXIS Axis 53 (id 53)
//     OtherSettings: AllowMotionCmdToSlave=true
//     encoder EncType=19
//       EncPara: MaxCount=#xffffffff
//     drive DrvType=16
//       DrvPara: MaxCount=#xffffffff
//         Analog: TorqueSetpointScale=10, ScaleFactorActTorque=0.1
//         TimeComp: TaskDelayCycles=1
//     controller CtrType=1
//       CtrPara: PriorControlFactor=1
//         Observer: BandWidth=20
//   AXIS Axis 54 (id 54)
//     OtherSettings: AllowMotionCmdToSlave=true
//     encoder EncType=19
//       EncPara: MaxCount=#xffffffff
//     drive DrvType=16
//       DrvPara: MaxCount=#xffffffff
//         Analog: TorqueSetpointScale=10, ScaleFactorActTorque=0.1
//         TimeComp: TaskDelayCycles=1
//     controller CtrType=1
//       CtrPara: PriorControlFactor=1
//         Observer: BandWidth=20
// I/O:
//   DEVICE Device 5 (NOV-DP-RAM)
//     Box 23 (Retain Handler)
//   DEVICE Device 1 (EtherCAT), AmsNetId 5.86.218.156.2.1
//     Term 51 (EK1200) [EK1200-5000 EtherCAT Power supply (2A E-Bus)]
//       Term 53 (EL6070-0033) [EL6070-0033 1Ch. Licence key terminal, individual licences]
//       Term 54 (EL1918) [EL1918, 8Ch. Safety Input 24V, TwinSAFE] (disabled)
//         modules: Module 1 (FSOE), Module 2 (FSLOGIC)
//       Term 55 (EL1918) [EL1918, 8Ch. Safety Input 24V, TwinSAFE] (disabled)
//         modules: Module 1 (FSOE), Module 2 (FSLOGIC)
//       Term 56 (EL1918) [EL1918, 8Ch. Safety Input 24V, TwinSAFE] (disabled)
//         modules: Module 1 (FSOE), Module 2 (FSLOGIC)
//       Term 57 (EL1918) [EL1918, 8Ch. Safety Input 24V, TwinSAFE] (disabled)
//         modules: Module 1 (FSOE), Module 2 (FSLOGIC)
//       Term 58 (EL1918) [EL1918, 8Ch. Safety Input 24V, TwinSAFE] (disabled)
//         modules: Module 1 (FSOE), Module 2 (FSLOGIC)
//       Term 59 (EL1918) [EL1918, 8Ch. Safety Input 24V, TwinSAFE] (disabled)
//         modules: Module 1 (FSOE), Module 2 (FSLOGIC)
//       Term 60 (EL1918) [EL1918, 8Ch. Safety Input 24V, TwinSAFE] (disabled)
//         modules: Module 1 (FSOE), Module 2 (FSLOGIC)
//       Term 61 (EL1918) [EL1918, 8Ch. Safety Input 24V, TwinSAFE] (disabled)
//         modules: Module 1 (FSOE), Module 2 (FSLOGIC)
//       Term 62 (EL9410) [EL9410 E-Bus Power Supplier  (Diagnostics)]
//       Term 63 (EL2904) [EL2904, 4 Ch. Safety Output 24V, 0.5A, TwinSAFE] (disabled)
//       Term 64 (EL2904) [EL2904, 4 Ch. Safety Output 24V, 0.5A, TwinSAFE] (disabled)
//         modules: Module 1 (FSOES), Module 2 (DO)
//       Term 65 (EL2904) [EL2904, 4 Ch. Safety Output 24V, 0.5A, TwinSAFE] (disabled)
//       Term 66 (EL2904) [EL2904, 4 Ch. Safety Output 24V, 0.5A, TwinSAFE] (disabled)
//       Term 67 (EL2904) [EL2904, 4 Ch. Safety Output 24V, 0.5A, TwinSAFE] (disabled)
//       Term 68 (EL2904) [EL2904, 4 Ch. Safety Output 24V, 0.5A, TwinSAFE] (disabled)
//       Term 69 (EL9410) [EL9410 E-Bus Power Supplier  (Diagnostics)]
//       Term 70 (EL1809) [EL1809 16Ch. Dig. Input 24V, 3ms]
//       Term 71 (EL1809) [EL1809 16Ch. Dig. Input 24V, 3ms]
//       Term 72 (EL1809) [EL1809 16Ch. Dig. Input 24V, 3ms]
//       Term 73 (EL2809) [EL2809 16Ch. Dig. Output 24V, 0.5A]
//       Term 74 (EL2809) [EL2809 16Ch. Dig. Output 24V, 0.5A]
//       Term 75 (EL2809) [EL2809 16Ch. Dig. Output 24V, 0.5A]
//       Term 76 (EL3162) [EL3162 2Ch. Ana. Input 0-10V]
//       Term 77 (EL4124) [EL4124 4Ch. Ana. Output 4-20mA, 16bit]
//       Term 78 (EL3154) [EL3154 4Ch. Ana. Input 4-20mA]
//       Term 79 (EK1110) [EK1110 EtherCAT extension]
//     Term 80 (EK1100) [EK1100 EtherCAT Coupler (2A E-Bus)]
//       Term 81 (EL7221-9014) [EL7221-9014 1Ch. MDP742 Servo motor output stage with OCT (50V, 8A RMS) and STO input]
//       Term 82 (EL9576) [EL9576 Bremschopper Klemme]
//       Term 83 (EL7221-9014) [EL7221-9014 1Ch. MDP742 Servo motor output stage with OCT (50V, 8A RMS) and STO input]
//       Term 84 (EL9576) [EL9576 Bremschopper Klemme]
//       Term 85 (EL7221-9014) [EL7221-9014 1Ch. MDP742 Servo motor output stage with OCT (50V, 8A RMS) and STO input]
//       Term 86 (EL9576) [EL9576 Bremschopper Klemme]
//       Term 87 (EL7221-9014) [EL7221-9014 1Ch. MDP742 Servo motor output stage with OCT (50V, 8A RMS) and STO input]
//       Term 88 (EL9576) [EL9576 Bremschopper Klemme]
//       Term 89 (EL7221-9014) [EL7221-9014 1Ch. MDP742 Servo motor output stage with OCT (50V, 8A RMS) and STO input]
//       Term 90 (EL9576) [EL9576 Brake chopper terminal]
//       Term 91 (EL7221-9014) [EL7221-9014 1Ch. MDP742 Servo motor output stage with OCT (50V, 8A RMS) and STO input]
//       Term 92 (EK1122) [EK1122 2 port EtherCAT junction]
//         Term 93 (EK1100) [EK1100 EtherCAT Coupler (2A E-Bus)]
//           Term 94 (EK1110) [EK1110 EtherCAT extension]
//         Drive 95 (C1150-DS-XC-1S) [C1150-DS-XC-1S V1.8b0]
//         Drive 96 (C1150-DS-XC-1S) [C1150-DS-XC-1S V1.8b0]
//         Drive 97 (C1150-DS-XC-1S) [C1150-DS-XC-1S V1.8b0]
//         Drive 98 (C1150-DS-XC-1S) [C1150-DS-XC-1S V1.8b0]
//         Drive 99 (C1150-DS-XC-1S) [C1150-DS-XC-1S V1.8b0]
//         Drive 100 (C1150-DS-XC-1S) [C1150-DS-XC-1S V1.8b0]
//         Drive 101 (C1150-DS-XC-1S) [C1150-DS-XC-1S V1.8b0]
//         Drive 102 (C1150-DS-XC-1S) [C1150-DS-XC-1S V1.8b0]
//         Drive 103 (C1150-DS-XC-1S) [C1150-DS-XC-1S V1.8b0]
//         Drive 104 (C1150-DS-XC-1S) [C1150-DS-XC-1S V1.8b0]
//         Drive 105 (C1150-DS-XC-1S) [C1150-DS-XC-1S V1.8b0]
//         Drive 106 (C1150-DS-XC-1S) [C1150-DS-XC-1S V1.8b0]
//         Drive 107 (C1150-DS-XC-1S) [C1150-DS-XC-1S V1.8b0]
//         Drive 108 (C1150-DS-XC-1S) [C1150-DS-XC-1S V1.8b0]
//         Drive 109 (C1150-DS-XC-1S) [C1150-DS-XC-1S V1.8b0]
//         Box 110 (EP6228-3032) [EP6228-3032 (IO Link Master Class B)]
//           modules: Module 1 (DeviceState Inputs Device), Module 2 (DeviceState Inputs), Module 3 (empty), Module 4 (empty), Module 5 (empty), Module 6 (empty), Module 7 (empty), Module 8 (empty), Module 9 (empty), Module 10 (empty)
//         Box 111 (EP6228-3032) [EP6228-3032 (IO Link Master Class B)]
//           modules: Module 1 (DeviceState Inputs Device), Module 2 (DeviceState Inputs), Module 3 (empty), Module 4 (empty), Module 5 (empty), Module 6 (empty), Module 7 (empty), Module 8 (empty), Module 9 (empty), Module 10 (empty)
//         Box 112 (EP6228-3032) [EP6228-3032 (IO Link Master Class B)]
//           modules: Module 1 (DeviceState Inputs Device), Module 2 (DeviceState Inputs), Module 3 (empty), Module 4 (empty), Module 5 (empty), Module 6 (empty), Module 7 (empty), Module 8 (empty), Module 9 (empty), Module 10 (empty)
//         Box 113 (EP6228-3032) [EP6228-3032 (IO Link Master Class B)]
//           modules: Module 1 (DeviceState Inputs Device), Module 2 (DeviceState Inputs), Module 3 (empty), Module 4 (empty), Module 5 (empty), Module 6 (empty), Module 7 (empty), Module 8 (empty), Module 9 (empty), Module 10 (empty)
//         Box 114 (EP6228-3032) [EP6228-3032 (IO Link Master Class B)]
//           modules: Module 1 (DeviceState Inputs Device), Module 2 (DeviceState Inputs), Module 3 (empty), Module 4 (empty), Module 5 (empty), Module 6 (empty), Module 7 (empty), Module 8 (empty), Module 9 (empty), Module 10 (empty)
//       Term 115 (EK1110) [EK1110 EtherCAT extension]
//     Drive 116 (C1150-DS-XC-1S) [C1150-DS-XC-1S V1.8b0]
//     Drive 117 (C1150-DS-XC-1S) [C1150-DS-XC-1S V1.8b0]
//     Drive 118 (C1150-DS-XC-1S) [C1150-DS-XC-1S V1.8b0]
//     Drive 119 (C1150-DS-XC-1S) [C1150-DS-XC-1S V1.8b0]
//     Drive 120 (C1150-DS-XC-1S) [C1150-DS-XC-1S V1.8b0]
//     Drive 121 (C1150-DS-XC-1S) [C1150-DS-XC-1S V1.8b0]
//     Box 122 (EP6228-3032) [EP6228-3032 (IO Link Master Class B)]
//       modules: Module 1 (DeviceState Inputs Device), Module 2 (DeviceState Inputs), Module 3 (empty), Module 4 (empty), Module 5 (empty), Module 6 (empty), Module 7 (empty), Module 8 (empty), Module 9 (empty), Module 10 (empty)
//     Box 123 (EP6228-3032) [EP6228-3032 (IO Link Master Class B)]
//       modules: Module 1 (DeviceState Inputs Device), Module 2 (DeviceState Inputs), Module 3 (empty), Module 4 (empty), Module 5 (empty), Module 6 (empty), Module 7 (empty), Module 8 (empty), Module 9 (empty), Module 10 (empty)
//     Box 124 (EP6228-3032) [EP6228-3032 (IO Link Master Class B)]
//       modules: Module 1 (DeviceState Inputs Device), Module 2 (DeviceState Inputs), Module 3 (empty), Module 4 (empty), Module 5 (empty), Module 6 (empty), Module 7 (empty), Module 8 (empty), Module 9 (empty), Module 10 (empty)
//     Box 125 (EP6228-3032) [EP6228-3032 (IO Link Master Class B)]
//       modules: Module 1 (DeviceState Inputs Device), Module 2 (DeviceState Inputs), Module 3 (empty), Module 4 (empty), Module 5 (empty), Module 6 (empty), Module 7 (empty), Module 8 (empty), Module 9 (empty), Module 10 (empty)
// variable links:
//   mover_demo/mover_demo Instance <-> Device 1 (EtherCAT)/Term 51 (EK1200)/Term 70 (EL1809)
//     Task_fileMan Inputs/IN.I000_ <-> Channel 1/Input
//     Task_fileMan Inputs/IN.I006_ <-> Channel 7/Input
//     Task_fileMan Inputs/IN.I007_ <-> Channel 8/Input
//     Task_fileMan Inputs/IN.I012_ <-> Channel 11/Input
//     Task_fileMan Inputs/IN.I013_ <-> Channel 12/Input
//     Task_fileMan Inputs/IN.I014_ <-> Channel 13/Input
//     Task_fileMan Inputs/IN.I015_ <-> Channel 14/Input
//     Task_fileMan Inputs/IN.I016_ <-> Channel 15/Input
//     Task_fileMan Inputs/IN.I017_ <-> Channel 16/Input
//     Task_fileMan Inputs/IN.I001_monitor_24V <-> Channel 2/Input
//     Task_fileMan Inputs/IN.I002_monitor_BR <-> Channel 3/Input
//     Task_fileMan Inputs/IN.I003_lufter_safety <-> Channel 4/Input
//     Task_fileMan Inputs/IN.I004_druckwachter_luftdruck_ok <-> Channel 5/Input
//     Task_fileMan Inputs/IN.I005_klimagerat_ok <-> Channel 6/Input
//     Task_fileMan Inputs/IN.I010_distanzsensor_verschmutzung_140_51 <-> Channel 9/Input
//     Task_fileMan Inputs/IN.I011_distanzsensor_verschmutzung_140_52 <-> Channel 10/Input
//   mover_demo/mover_demo Instance <-> Device 1 (EtherCAT)/Term 51 (EK1200)/Term 71 (EL1809)
//     Task_fileMan Inputs/IN.I020_ultraschall_bereit_150_20 <-> Channel 1/Input
//     Task_fileMan Inputs/IN.I024_ultraschall_bereit_155_20 <-> Channel 5/Input
//     Task_fileMan Inputs/IN.I021_ultraschall_fehler_150_20 <-> Channel 2/Input
//     Task_fileMan Inputs/IN.I025_ultraschall_fehler_155_20 <-> Channel 6/Input
//     Task_fileMan Inputs/IN.I022_ultraschall_us_on_150_20 <-> Channel 3/Input
//     Task_fileMan Inputs/IN.I026_ultraschall_us_on_155_20 <-> Channel 7/Input
//     Task_fileMan Inputs/IN.I023_ultraschall_nullpos_150_20 <-> Channel 4/Input
//     Task_fileMan Inputs/IN.I027_ultraschall_nullpos_155_20 <-> Channel 8/Input
//     Task_fileMan Inputs/IN.I030_rfid_test_link_out1_170_20 <-> Channel 9/Input
//     Task_fileMan Inputs/IN.I031_rfid_test_link_out2_170_20 <-> Channel 10/Input
//     Task_fileMan Inputs/IN.I032_rfid_test_link_out3_170_20 <-> Channel 11/Input
//     Task_fileMan Inputs/IN.I033_rfid_test_link_out1_170_21 <-> Channel 12/Input
//     Task_fileMan Inputs/IN.I034_rfid_test_link_out2_170_21 <-> Channel 13/Input
//     Task_fileMan Inputs/IN.I035_rfid_test_link_out3_170_21 <-> Channel 14/Input
//     Task_fileMan Inputs/IN.I036_ <-> Channel 15/Input
//     Task_fileMan Inputs/IN.I037_ <-> Channel 16/Input
//   mover_demo/mover_demo Instance <-> Device 5 (NOV-DP-RAM)/Box 23 (Retain Handler)
//     PlcTask Retains/PERS.iRecipeCurrent <-> Retains/PERS.iRecipeCurrent_[851]
//     PlcTask Retains/PERS.iStationTimeDef1 <-> Retains/PERS.iStationTimeDef1_[851]
//     PlcTask Retains/PERS.iStationTimeDef2 <-> Retains/PERS.iStationTimeDef2_[851]
//     PlcTask Retains/PERS.udiCount6Mauto <-> Retains/PERS.udiCount6Mauto_[851]
//     PlcTask Retains/PERS.udiCount6Mon <-> Retains/PERS.udiCount6Mon_[851]
//     PlcTask Retains/PERS.udiCountHauto <-> Retains/PERS.udiCountHauto_[851]
//     PlcTask Retains/PERS.udiCountHon <-> Retains/PERS.udiCountHon_[851]
//     PlcTask Retains/PERS.udiTempNOK <-> Retains/PERS.udiTempNOK_[851]
//     PlcTask Retains/PERS.udiTempOK <-> Retains/PERS.udiTempOK_[851]
//   mover_demo/mover_demo Instance <-> NC-Task 1 SAF/Axes/SIMU_ST145_01Y
//     Task_fileMan Inputs/SIMU.axis_ref[18].NcToPlc <-> Outputs/ToPlc
//     Task_fileMan Outputs/SIMU.axis_ref[18].PlcToNc <-> Inputs/FromPlc
//   mover_demo/mover_demo Instance <-> NC-Task 1 SAF/Axes/SIMU_ST145_02Z
//     Task_fileMan Inputs/SIMU.axis_ref[19].NcToPlc <-> Outputs/ToPlc
//     Task_fileMan Outputs/SIMU.axis_ref[19].PlcToNc <-> Inputs/FromPlc
//   mover_demo/mover_demo Instance <-> NC-Task 1 SAF/Axes/ST110_01Y
//     PlcTask Inputs/ST110_Axis.axis110_01Y.axis.NcToPlc <-> Outputs/ToPlc
//     PlcTask Outputs/ST110_Axis.axis110_01Y.axis.PlcToNc <-> Inputs/FromPlc
//   mover_demo/mover_demo Instance <-> NC-Task 1 SAF/Axes/ST110_02Z
//     PlcTask Inputs/ST110_Axis.axis110_02Z.axis.NcToPlc <-> Outputs/ToPlc
//     PlcTask Outputs/ST110_Axis.axis110_02Z.axis.PlcToNc <-> Inputs/FromPlc
//   mover_demo/mover_demo Instance <-> NC-Task 1 SAF/Axes/ST110_03Z
//     PlcTask Inputs/ST110_Axis.axis110_03Z.axis.NcToPlc <-> Outputs/ToPlc
//     PlcTask Outputs/ST110_Axis.axis110_03Z.axis.PlcToNc <-> Inputs/FromPlc
//   mover_demo/mover_demo Instance <-> NC-Task 1 SAF/Axes/ST110_04Z
//     PlcTask Inputs/ST110_Axis.axis110_04Z.axis.NcToPlc <-> Outputs/ToPlc
//     PlcTask Outputs/ST110_Axis.axis110_04Z.axis.PlcToNc <-> Inputs/FromPlc
//   mover_demo/mover_demo Instance <-> NC-Task 1 SAF/Axes/ST110_10W
//     PlcTask Inputs/ST110_Axis.axis110_10W.axis.NcToPlc <-> Outputs/ToPlc
//     PlcTask Outputs/ST110_Axis.axis110_10W.axis.PlcToNc <-> Inputs/FromPlc
//   mover_demo/mover_demo Instance <-> NC-Task 1 SAF/Axes/ST115_01Y
//     PlcTask Inputs/ST115_Axis.axis115_01Y.axis.NcToPlc <-> Outputs/ToPlc
//     PlcTask Outputs/ST115_Axis.axis115_01Y.axis.PlcToNc <-> Inputs/FromPlc
//   mover_demo/mover_demo Instance <-> NC-Task 1 SAF/Axes/ST115_02Z
//     PlcTask Inputs/ST115_Axis.axis115_02Z.axis.NcToPlc <-> Outputs/ToPlc
//     PlcTask Outputs/ST115_Axis.axis115_02Z.axis.PlcToNc <-> Inputs/FromPlc
//   mover_demo/mover_demo Instance <-> NC-Task 1 SAF/Axes/ST115_03Z
//     PlcTask Inputs/ST115_Axis.axis115_03Z.axis.NcToPlc <-> Outputs/ToPlc
//     PlcTask Outputs/ST115_Axis.axis115_03Z.axis.PlcToNc <-> Inputs/FromPlc
//   mover_demo/mover_demo Instance <-> NC-Task 1 SAF/Axes/ST115_10W
//     PlcTask Inputs/ST115_Axis.axis115_10W.axis.NcToPlc <-> Outputs/ToPlc
//     PlcTask Outputs/ST115_Axis.axis115_10W.axis.PlcToNc <-> Inputs/FromPlc
//   mover_demo/mover_demo Instance <-> NC-Task 1 SAF/Axes/ST120_01Y
//     PlcTask Inputs/ST120_Axis.axis120_01Y.axis.NcToPlc <-> Outputs/ToPlc
//     PlcTask Outputs/ST120_Axis.axis120_01Y.axis.PlcToNc <-> Inputs/FromPlc
//   mover_demo/mover_demo Instance <-> NC-Task 1 SAF/Axes/ST120_02Z
//     PlcTask Inputs/ST120_Axis.axis120_02Z.axis.NcToPlc <-> Outputs/ToPlc
//     PlcTask Outputs/ST120_Axis.axis120_02Z.axis.PlcToNc <-> Inputs/FromPlc
//   mover_demo/mover_demo Instance <-> NC-Task 1 SAF/Axes/ST125_01Y
//     PlcTask Inputs/ST125_Axis.axis125_01Y.axis.NcToPlc <-> Outputs/ToPlc
//     PlcTask Outputs/ST125_Axis.axis125_01Y.axis.PlcToNc <-> Inputs/FromPlc
//   mover_demo/mover_demo Instance <-> NC-Task 1 SAF/Axes/ST125_02Z
//     PlcTask Inputs/ST125_Axis.axis125_02Z.axis.NcToPlc <-> Outputs/ToPlc
//     PlcTask Outputs/ST125_Axis.axis125_02Z.axis.PlcToNc <-> Inputs/FromPlc
//   mover_demo/mover_demo Instance <-> NC-Task 1 SAF/Axes/ST125_10W
//     PlcTask Inputs/ST125_Axis.axis125_10W.axis.NcToPlc <-> Outputs/ToPlc
//     PlcTask Outputs/ST125_Axis.axis125_10W.axis.PlcToNc <-> Inputs/FromPlc
//   mover_demo/mover_demo Instance <-> NC-Task 1 SAF/Axes/ST145_01Y
//     PlcTask Inputs/ST145_Axis.axis145_01Y.axis.NcToPlc <-> Outputs/ToPlc
//     PlcTask Outputs/ST145_Axis.axis145_01Y.axis.PlcToNc <-> Inputs/FromPlc
//   mover_demo/mover_demo Instance <-> NC-Task 1 SAF/Axes/ST145_02Z
//     PlcTask Inputs/ST145_Axis.axis145_02Z.axis.NcToPlc <-> Outputs/ToPlc
//     PlcTask Outputs/ST145_Axis.axis145_02Z.axis.PlcToNc <-> Inputs/FromPlc
//   mover_demo/mover_demo Instance <-> NC-Task 1 SAF/Axes/ST145_10W
//     PlcTask Inputs/ST145_Axis.axis145_10W.axis.NcToPlc <-> Outputs/ToPlc
//     PlcTask Outputs/ST145_Axis.axis145_10W.axis.PlcToNc <-> Inputs/FromPlc
//   mover_demo/mover_demo Instance <-> NC-Task 1 SAF/Axes/ST180_01Y
//     PlcTask Inputs/ST180_Axis.axis180_01Y.axis.NcToPlc <-> Outputs/ToPlc
//     PlcTask Outputs/ST180_Axis.axis180_01Y.axis.PlcToNc <-> Inputs/FromPlc
//   mover_demo/mover_demo Instance <-> NC-Task 1 SAF/Axes/ST180_02Z
//     PlcTask Inputs/ST180_Axis.axis180_02Z.axis.NcToPlc <-> Outputs/ToPlc
//     PlcTask Outputs/ST180_Axis.axis180_02Z.axis.PlcToNc <-> Inputs/FromPlc
//   mover_demo/mover_demo Instance <-> NC-Task 1 SAF/Axes/ST180_10Z
//     PlcTask Inputs/ST180_Axis.axis180_10Z.axis.NcToPlc <-> Outputs/ToPlc
//     PlcTask Outputs/ST180_Axis.axis180_10Z.axis.PlcToNc <-> Inputs/FromPlc

CONFIGURATION mover_demo
    RESOURCE PLC ON TwinCAT3
        TASK PlcTask(INTERVAL := T#10ms, PRIORITY := 20);
        TASK VISU_TASK(INTERVAL := T#10ms, PRIORITY := 21);
        PROGRAM MAIN WITH PlcTask : MAIN;
        PROGRAM TruMark_Ethercat WITH PlcTask : TruMark_Ethercat;
        PROGRAM TruMark_SingleCmds WITH PlcTask : TruMark_SingleCmds;
        PROGRAM VisuElems_Visu_Prg WITH VISU_TASK : VisuElems.Visu_Prg;
    END_RESOURCE
END_CONFIGURATION

// ---- DUTs/Helptec/Axis/AxisBase_t.TcDUT
TYPE ABSTRACT AxisBase_t :
STRUCT
    rActPos : REAL; // Current position
    bInPos  : SINT; // Current position index, 99=unknown
END_STRUCT
END_TYPE

// ---- DUTs/Helptec/Axis/AxisBeckhoff_t.TcDUT
TYPE AxisBeckhoff_t EXTENDS AxisBase_t :
STRUCT
    axis : AXIS_REF; // reference of the axis 
END_STRUCT
END_TYPE

// ---- DUTs/Helptec/Axis/AxisLinMot_t.TcDUT
TYPE AxisLinMot_t EXTENDS AxisBeckhoff_t :
STRUCT
    bCtrlHi AT %Q* : BYTE; // Axis control word, Hi-Byte
    wState  AT %I* : WORD; // Axis status word
END_STRUCT
END_TYPE

// ---- DUTs/Helptec/Axis/typeInputArea.TcDUT
TYPE typeInputArea :
STRUCT
	SigAllToTheInpPor: UINT;
      	ControllerInformationFlag: UINT;
      	CurrentPosition : DINT;
      	CurrentSpeed : UINT;
      	CurrentPushForce : UINT;
      	TargetPosition : DINT;
      	Alarm1 : USINT;
      	Alarm2 : USINT;
      	Alarm3 : USINT;
      	Alarm4 : USINT;
END_STRUCT
END_TYPE

// ---- DUTs/Helptec/Axis/typeOutputArea.TcDUT
TYPE typeOutputArea :
STRUCT
    OutPorToWhiSigAreAll : UINT;
    NumericalDataFlag    : UINT;
    StartFlag            : USINT;
    OperationMethod      : USINT;
    Speed                : UINT;
    TargetPosition       : DINT;
    Acceleration         : UINT;
    Deceleration         : UINT;
    PushingForce         : UINT;
    TriggerLv            : UINT;
    PushingSpeed         : UINT;
    PushingForceForPos   : UINT;
    Area1                : DINT;
    Area2                : DINT;
    PositioningWidth     : DINT;
END_STRUCT
END_TYPE

// ---- DUTs/Helptec/Cylinder2Pos_config.TcDUT
TYPE Cylinder2Pos_config :
STRUCT
    toGS_alarm_time : DINT; // maximum time allowed to go from AS to GS
    toAS_alarm_time : DINT; // maximum time allowed to go from GS to AS
    toGS_wait_time  : DINT; // additionnal waiting time, added when GS sensor is reached
    toAS_wait_time  : DINT; // additionnal waiting time, added when AS sensor is reached
END_STRUCT
END_TYPE

// ---- DUTs/Helptec/Recipe/RecipeAxisLinear2Pos_t.TcDUT
TYPE RecipeAxisLinear2Pos_t :
STRUCT
    rPosGS    : REAL;
    rPosAS    : REAL;
    rVeloToAS : REAL;
    rVeloToGS : REAL;
    rAccel    : REAL;
    rDecel    : REAL;
    rJerk     : REAL;
END_STRUCT
END_TYPE

// ---- DUTs/Helptec/RS_Axis/MoveProfile1D_t.TcDUT
// Specify a 1D mouvement, the position only represents a point in the 1D space
TYPE MoveProfile1D_t EXTENDS MoveProfile_t:
STRUCT
    lrPosition  : LREAL;         // Position to go
END_STRUCT
END_TYPE

// ---- DUTs/Helptec/RS_Axis/MoveProfile_t.TcDUT
// A move profile only provide velocity and its derivatives
TYPE MoveProfile_t :
STRUCT
    lrVelocity  : REAL;         // Velocity to position
    lrAccel     : REAL;         // acceleration to position
    lrDecel     : REAL;         // deceleration to position
    lrJerk      : REAL;         // jerk to position
END_STRUCT
END_TYPE

// ---- DUTs/Helptec/RS_Axis/TriggerType_e.TcDUT
// Tell when the 'InRange' signal should be true
// The trigger permit your application to run faster by allowing
// another element/axis to start moving before the movement is really
// completed
{attribute 'qualified_only'}
{attribute 'strict'}
TYPE TriggerType_e :
(
    None := 0,     // no trigger is used. The InRange flag will raise at the same moment as the 'InPos' flag
    SetPos := 1,   // The trigger is set at the given position
    FromLast := 2, // The trigger is placed relative to the last position
    FromEnd := 3,  // The trigger is placed relative to end position
    _max
);
END_TYPE

// ---- DUTs/Helptec/RS_Axis/VectorMove1D_t.TcDUT
// Configuration structure for a VectorMove1D
// This configuration is typically stored inside a ricipies
TYPE VectorMove1D_t :
STRUCT
    lrVelocity  : REAL;  // Velocity to position
    lrAccel     : REAL;  // acceleration to position
    lrDecel     : REAL;  // deceleration to position
    lrJerk      : REAL;  // jerk to position
    lrPosition  : LREAL; // Position to go
    TriggerType : INT;   // the kind of trigger used
    TriggerPos  : LREAL; // trigger position, ignore if TriggerType is None
    Timeout_ms  : DINT;  // timeout value for this movement vector expressed in milisecond
END_STRUCT
END_TYPE

// ---- DUTs/Helptec/structButton.TcDUT
TYPE structButton :
STRUCT
	button	:	BOOL;	// BUTTON SIGNAL FROM HMI
	disable	:	BOOL;	// FORCE BUTTON INACTIV
	rtrig	:	BOOL;	// RISING EDGE
	ftrig	:	BOOL;	// FALLING EDGE
	press	:	BOOL;	// BUTTON PRESSED
	on		:	BOOL;	// FUNCTION ON (GREEN)
	error	:	BOOL;	// FUNCTION ERROR (RED)
END_STRUCT
END_TYPE

// ---- POUs/20_AUTO/Axis_e.TcTLEO
{attribute 'qualified_only'}
{attribute 'strict'}
{attribute 'to_string'}
TYPE Axis_e :
(
    ST110_01Y,  //  0
    ST110_02Z,  //  1
    ST110_03Z,  //  2
    ST110_04Z,  //  3
	ST110_10W,  //  4
    ST115_01Y,  //  5
    ST115_02Z,  //  6
    ST115_03Z,  //  7
    ST115_04Z,  //  8
	ST115_10W,  //  9
    ST120_01Y,  // 10
    ST120_02Z,  // 11
    ST125_01Y,  // 12
    ST125_02Z,  // 13
	ST125_10W,  // 14
	ST130_01Z,  // 15
	ST130_10Z,  // 16
	ST135_01Z,  // 17
	ST135_10Z,  // 18
	ST145_01Y,  // 19
	ST145_02Z,  // 20
	ST145_10W,  // 21
	ST160_01Z,  // 22
	ST165_01Z,  // 23
	ST170_01Z,  // 24
	ST180_01Y,  // 25
	ST180_02Z,  // 26
	ST180_10Z,  // 27
	ST185_01Y,  // 28
	ST185_02Z,  // 29
	ST185_10Z,  // 30
    _max
);
END_TYPE

// ---- POUs/20_AUTO/BuR SuperTrack com/CT_Shuttle_BR_to_Tc_Status_t.TcDUT
{attribute 'pack_mode' := '1'}
TYPE
CT_Shuttle_BR_to_Tc_Status_t :
STRUCT
    {STweep.disable}
    reserve1               : BIT; // 
    recovering             : BIT; // 
    at_target              : BIT; // 
    in_position            : BIT; // 
    servo_enabled          : BIT; // 
    moving_to_load_target  : BIT; // 
    lost_position_feedback : BIT; // 
    reserve8               : BIT; // 
    {STweep.Enable}
END_STRUCT
END_TYPE

// ---- POUs/20_AUTO/BuR SuperTrack com/CT_Shuttle_BR_to_Tc_t.TcDUT
{attribute 'pack_mode' := '1'}
TYPE
CT_Shuttle_BR_to_Tc_t :
STRUCT
    bStatus             : CT_Shuttle_BR_to_Tc_Status_t; // status flag	
    diCurrentPos_um     : DINT;                         // current position, expressed as um
    iCurrentVelo_mmps   : INT;                          // current velocity in mm per second
    bDestinationStation : BYTE;                         // 0 = no station, else the destination station
    bShelfLentgh_mm     : INT;                          // shelf length in mm 
END_STRUCT
END_TYPE

// ---- POUs/20_AUTO/BuR SuperTrack com/CT_Shuttle_BR_to_Tc_u.TcDUT
{attribute 'pack_mode' := '1'}
TYPE
CT_Shuttle_BR_to_Tc_u :
UNION
    asStruct : ARRAY[1..20] OF CT_Shuttle_BR_to_Tc_t;
    asArray  : ARRAY[0..20 * SIZEOF(CT_Shuttle_BR_to_Tc_t) - 1] OF USINT;
END_UNION
END_TYPE

// ---- POUs/20_AUTO/BuR SuperTrack com/CT_Shuttle_Tc_To_BR_Command_t.TcDUT
{attribute 'pack_mode' := '1'}
TYPE CT_Shuttle_Tc_To_BR_Command_t :
STRUCT
    release        : BIT; // Move the shuttle to the next position
    dirFarward     : BIT; // Specify the farward direction (depends on the SuperTrak configuration)
    dirReverse     : BIT; // Specify the reverse direction (depends on the SuperTrak configuration) 
    echo_in_pos    : BIT; // Echo signal for the In Position signal, this is to ensure the flag In Pos is not missed
    echo_at_target : BIT; // Echo signal for the At target signal, this is to ensure the flag At target is not missed
    reserve6       : BIT; // 
    reserve7       : BIT; // 
    reserve8       : BIT; // 
END_STRUCT
END_TYPE

// ---- POUs/20_AUTO/BuR SuperTrack com/CT_Shuttle_Tc_to_BR_t.TcDUT
TYPE CT_Shuttle_Tc_to_BR_t :
STRUCT
    bCommand     : BYTE; (* command bit field *)
    bNextStation : BYTE; (* next station *)
    iNextOffset  : INT;  (* needs to be between -500 and 500 *)
END_STRUCT
END_TYPE

// ---- POUs/20_AUTO/BuR SuperTrack com/CT_Shuttle_Tc_to_BR_u.TcDUT
TYPE CT_Shuttle_Tc_to_BR_u :
UNION
    asStruct : ARRAY[1..20] OF CT_Shuttle_Tc_to_BR_t;
    asArray  : ARRAY[0..200] OF USINT;
END_UNION
END_TYPE

// ---- POUs/20_AUTO/BuR SuperTrack com/CT_Track_BR_to_TC_Status_t.TcDUT
// track status from BR to Twincat
{attribute 'pack_mode' := '1'}
TYPE CT_Track_BR_to_TC_Status_t :
STRUCT
    ready                 : BIT; // The track is ready to take commands
    error                 : BIT; // The track is in error
    powerOn               : BIT; // The shuttles are energized
    inOperation           : BIT; // The track is now under control of CleverTrackLib
    allIdSet              : BIT; // All the ID's are set and verified
    unknownMoverAtTarget1 : BIT; // Tell TC that the shuttle is at the first target ready to take order
    reserve7              : BIT; // 
    reserve8              : BIT; // 
END_STRUCT
END_TYPE

// ---- POUs/20_AUTO/BuR SuperTrack com/CT_Track_BR_to_Tc_t.TcDUT
TYPE CT_Track_BR_to_Tc_t :
STRUCT
    bStatus : CT_Track_BR_to_TC_Status_t;
    diError : DINT;
END_STRUCT
END_TYPE

// ---- POUs/20_AUTO/BuR SuperTrack com/CT_Track_BR_to_Tc_u.TcDUT
{attribute 'pack_mode' := '1'}
TYPE CT_Track_BR_to_Tc_u :
UNION
    asStruct : CT_Track_BR_to_Tc_t;
    asArray  : ARRAY[0..SIZEOF(CT_Track_BR_to_Tc_t)-1] OF USINT;
END_UNION
END_TYPE

// ---- POUs/20_AUTO/BuR SuperTrack com/CT_Track_Tc_to_BR_Command_t.TcDUT
// track command from twincat to BR PLC
{attribute 'pack_mode' := '1'}
TYPE CT_Track_Tc_to_BR_Command_t :
STRUCT
    {STweep.disable}
    twincatReady                : BIT; // TRUE when the twincat PLC is ready to operate (not in error and cleverTrackLib is ok)
    wholePathFree               : BIT; // TRUE wen all the station are in a position where all the mover can freely rotate on all the track
    resetErrors                 : BIT; // rising edge of this signal will reset all current errors from the supertrack
    enablePower                 : BIT; // enable power on the track, this will energized all shuttles and they will stay at current place
    enableProcess               : BIT; // allow cleverTrackLib to take control of the release sequence
    startMoverNumberingSequence : BIT; // tell BR PLC that we will start the number attribution sequence
    setShuttleNumber            : BIT; // tell BR PLC that we will give the next available number to the current shuttle
    releaseUnknownShuttle       : BIT; // tell BR PLC that we will pass this shuttle without attributing it a number
	{STweep.Enable}
END_STRUCT
END_TYPE

// ---- POUs/20_AUTO/BuR SuperTrack com/CT_Track_Tc_to_BR_t.TcDUT
TYPE CT_Track_Tc_to_BR_t :
STRUCT
    bCommand : BYTE; (* command bit field for the track system *)
END_STRUCT
END_TYPE

// ---- POUs/20_AUTO/BuR SuperTrack com/CT_Track_Tc_to_BR_u.TcDUT
TYPE CT_Track_Tc_to_BR_u :
UNION
    asStruct : CT_Track_Tc_to_BR_t;
    asArray  : ARRAY[0..SIZEOF(CT_Track_Tc_to_BR_t)-1] OF USINT;
END_UNION
END_TYPE

// ---- POUs/20_AUTO/LinearAxis_e.TcTLEO
{attribute 'qualified_only'}
TYPE LinearAxis_e :
(
    ST105_11Z, //0
    ST110_01Y,
    ST110_02Z,
    ST110_03Z,
    ST110_04Z,
    ST115_01Y,	//5
    ST115_02Z,
    ST115_03Z,
    ST115_04Z,
    ST120_01Y,
    ST120_02Z,	//10
    ST125_01Y,
    ST125_02Z,
	ST130_01Z,
	ST130_10Z,
	ST135_01Z,	//15
	ST135_10Z,
	ST145_01Y,
	ST145_02Z,
	ST160_01Z,
	ST165_01Z,	//20
	ST170_01Z,
	ST180_01Y,
	ST180_02Z,
	ST180_10Z,
	ST185_01Y,	//25
	ST185_02Z,
	ST185_10Z,
    _max
);
END_TYPE

// ---- POUs/20_AUTO/RecipeType_e.TcTLEO
{attribute 'qualified_only'}
{attribute 'strict'}
TYPE RecipeType_e :
(
    Smart := 0,
    Pro := 1,
    Mini := 2,
    // Smart_Kristall := 3,
    // Pro_Smart := 4,
    // Pro_Blue := 5,
    // Pro_Smart_Kristall := 6,
    // Pro_Smart_Maxi := 7,
    // Pro_Smart_Maxi_Kristall := 8,
    _max
);
END_TYPE

// ---- POUs/20_AUTO/Mover/ApproachScenario_e.TcTLEO
{attribute 'qualified_only'}
{attribute 'strict'}
{attribute 'to_string'}
TYPE
ApproachScenario_e :
(
    WaitOnFinishedProcess,
    WaitOnFreeStation,
    DoNotWait,
    WaitOnPrevProcess,
    WaitOnExternalTrigger,
    _MAX
);
END_TYPE

// ---- POUs/20_AUTO/Mover/MoverDirection_e.TcTLEO
{attribute 'qualified_only'}
{attribute 'strict'}
TYPE MoverDirection_e :
(
	Farward,
	Reverse
);
END_TYPE

// ---- POUs/20_AUTO/Mover/MoverState_e.TcTLEO
{attribute 'qualified_only'}
{attribute 'strict'}
{attribute 'to_string'}
TYPE
MoverState_e :
(
    OperationDone,       // The operation on the mover is done, a new station needs to be given
    WaitOnNextStation,   // wait on the next station to be ready. The waiting depend on the scenario of the next station
    MovingToStation,     // the mover is moving or try to move to the next station
    InStationPos,        // The mover is currently at the station position (aka target pos.), waiting on the process to begin
    InOperation,         // The attached process of the mover is running. The mover is not able to move
    PerformRelativeMove, // Moving the mover when already in operation, go to WaitRelativeMoveEnd when mover actually moving
    WaitRelativeMoveEnd, // Wait on the At_pos flag
    _MAX
);
END_TYPE

// ---- POUs/20_AUTO/Mover/StationName_e.TcTLEO
{attribute 'qualified_only'}
{attribute 'strict'}
{attribute 'to_string'}
TYPE
StationName_e :
(
    Station100 := 1,
    Station110 := 2,
    Station120 := 3,
    Station130 := 4,
    Station140 := 5,
    Station150 := 6,
    Station160 := 7,
    Station170 := 8,
    Station180 := 9,
    Station190 := 10,
    Station200 := 11,
    Station210 := 12,
    Station220 := 13,
    Station230 := 14,
    Station240 := 15,
    Station250 := 16,
    Station260 := 17,
    Station270 := 18
);
END_TYPE

// ---- POUs/20_AUTO/Recipe_21_101_t.TcDUT
// Recipe for the 21.101 machine
TYPE Recipe_21_101_t :
STRUCT
    linearAxis     : ARRAY[0..LinearAxis_e._max - 1] OF LinearMotionMan_Config_t;
    cylinder2Pos   : ARRAY[0..StationList_e._max] OF ARRAY[0..CONST.MAX_CYLINDER_PER_STATION] OF Cylinder2Pos_config;
    stationOffsets : ARRAY[0..CONST.STATION_NUMBER - 1] OF REAL;
    st105          : ST105_Recipe_t;
    st110          : ST110_Recipe_t;
    st115          : ST115_Recipe_t;
    st120          : ST120_Recipe_t;
    st125          : ST125_Recipe_t;
    st128          : ST128_Recipe_t;
    st130          : ST130_Recipe_t;
    st140          : ST140_Recipe_t;
    st145          : ST145_Recipe_t;
    st150          : ST150_Recipe_t;
    st160          : ST160_Recipe_t;
    st165          : ST160_Recipe_t;
    st170          : ST170_Recipe_t;
    st175          : ST175_Recipe_t;
    st180          : ST180_Recipe_t;
    st185          : ST185_Recipe_t;
END_STRUCT
END_TYPE

// ---- POUs/20_AUTO/ST100/ST100_Laser_e.TcTLEO
{attribute 'qualified_only'}
{attribute 'strict'}
TYPE ST100_Laser_e :
(
    RESET := 0,               // Reset
    INIT := 100,              // Initialisieren 
    READY := 999,             // READY to Start, Init Done 
    START := 1000,            // Start Zyklisch
    MOVER_FREE_OP,            // Ab here, operation without mover can be done
    waitOnMover,              // wait until the mover is there
    MOVER_NEEDED_OP,          // Ab here, a mover in position is needed to perform the action
    proceedOperation_1,       // proceed to some operation
    move_mover_to_next_piece, // move the mover to the next piece if needed
    proceedOperation_2,       // proceed to some operation
    SYNC_MOVER_LEAVE,         // MoverMan need to take the mover
    DONE := 8000,             // Ablauf beendet 
    ERROR := 9000,            // Fehler 
    _max
);
END_TYPE

// ---- POUs/20_AUTO/ST105/Fanuc_robot/Fanuc_command_std_to_robot_t.TcDUT
{attribute 'pack_mode' := '1'}
TYPE Fanuc_command_std_to_robot_t :
STRUCT
    IMDSTP          : BIT; // Stopp sofort
    Hold            : BIT; // Stopp
    SFSPD           : BIT; // Sicher Geschwindigkeit
    Abort_CycleStop : BIT; // Progfamm abrechen/Zyklus ende
    FaultReset      : BIT; // Fehler Rücksetzten
    Start           : BIT; // Start nach CycleEnd / Pause
    Home            : BIT; // Fahrt zur Homposition !
    Enable          : BIT; // Bereit
END_STRUCT
END_TYPE

// ---- POUs/20_AUTO/ST105/Fanuc_robot/ST105_Fanuc_command_t.TcDUT
TYPE ST105_Fanuc_command_t :
STRUCT
    FG_Pick          : BIT; // Pick pieces at the feeder side
    FG_Place         : BIT; // Place pieces at the mover side
    Cycle_end        : BIT; // Tell the robot to stop working and go full up when finished
    One_cycle        : BIT; // Tell the robot to do just one cycleand and go full up when finished
    Use_griper_left  : BIT; // Use the left griper
    Use_griper_right : BIT; // Use the right griper
    reserve_b6       : BIT; // 
    reserve_b7       : BIT; // 
    ZOff             : BIT; // negative flag for the Z offset
    XOff             : BIT; // negative flag for the X offset
    YOff             : BIT; // negative flag for the Y offset
    reserve_b11      : BIT; // 
    reserve_b12      : BIT; // 
    reserve_b13      : BIT; // 
    reserve_b14      : BIT; // 
    reserve_b15      : BIT; // 
END_STRUCT
END_TYPE

// ---- POUs/20_AUTO/ST105/Fanuc_robot/ST105_Fanuc_status_t.TcDUT
TYPE ST105_Fanuc_status_t :
STRUCT
    Picked         : BIT; // Piece(s) picked by the robot
    Placed         : BIT; // Piece(s) placed by the robot
    Ready_to_pick  : BIT; // Robot is in pick position
    Ready_to_place : BIT; // Robot is in place position
    reserve_b4     : BIT; // 
    reserve_b5     : BIT; // 
    reserve_b6     : BIT; // 
    reserve_b7     : BIT; // 
END_STRUCT
END_TYPE

// ---- POUs/20_AUTO/ST105/ST105_PnpVerPushPos_e.TcDUT
{attribute 'qualified_only'}
{attribute 'strict'}
TYPE ST105_PnpVerPushPos_e :
(
	down,
	up,
	_max
);
END_TYPE

// ---- POUs/20_AUTO/ST105/ST105_Recipe_t.TcDUT
TYPE ST105_Recipe_t :
STRUCT
    xUseVerLeft        : BOOL; // Is the left vertical picker element is used
    xUseVerRight       : BOOL; // Is the right vertical picker element is used
    FeederConfig       : FeederDelays_t;
    FeederSize         : DINT;  // tell the feeder slots number, if it has 2 slots or 
    RotaryTableOffset  : LREAL; // feeder offset
    PickOffset_X_deci  : UINT;  // X offset of picking position
    PickOffset_Y_deci  : UINT;  // Y offset of picking position
    PickUpPos_Z_deci   : UINT;  // Z traveling height from pick to place position
    isPickOffset_X_neg : BOOL;  // tell the robot that PickOffset_X_deci is negative
    isPickOffset_Y_neg : BOOL;  // tell the robot that PickOffset_Y_deci is negative
    isPickUpPos_Z_neg  : BOOL;  // tell the robot that PickUpPos_Z_deci is negative
END_STRUCT
END_TYPE

// ---- POUs/20_AUTO/ST105/ST105_Feeder_e.TcDUT
{attribute 'qualified_only'}
{attribute 'strict'}
TYPE ST105_Feeder_e :
(
    RESET := 0, // Reset

    INIT := 100, // Initialisieren 
    Init_home_table,
    Init_simu_home_table,
    Init_table_go_to_zero,
    Init_reset_search_index,
    Init_set_table_pos,
    Init_see_if_piece_there,
	Init_apply_feeder_offset, // If homing screw are not placed exactly at the same place, we fix that here

    READY := 999,  // READY to Start, Init Done 
    START := 1000, // Start Zyklisch
    check_if_feeding_necessary,
	wait_on_a_piece,
	load_piece,

    DONE := 8000,  // Ablauf beendet 
    ERROR := 9000, // Fehler 
    _max
);
END_TYPE

// ---- POUs/20_AUTO/ST105/ST105_Pnp_e.TcTLEO
{attribute 'qualified_only'}
{attribute 'strict'}
{attribute 'to_string'}
TYPE
ST105_Pnp_e :
(
    RESET := 0, // Reset

    INIT := 100, // Initialisieren 
    Init_HomeVertical,
    Init_VerticalDown,
    Init_RobotRaiseStartFlag,
    Init_RobotFallStartFlag,
    Init_check_if_pces_handled,

    READY := 999,  // READY to Start, Init Done 
    START := 1000, // Start Zyklisch
    MOVER_FREE_OP, // Ab here, operation without mover can be done

    wait_on_feeder, // wait on feeder to be ready
    push_up_casing, // push up the casing (gehäuse)
    Robot_Pick,     // send pick signal to the robot
    Robot_wait_picked_falling,
    pusher_down,

    waitOnMover,     // wait until the mover is there
    MOVER_NEEDED_OP, // Since here, a mover in position is needed to perform the action

    Robot_place, // send place signal to the robot
    Robot_wait_placed_falling,

    SYNC_MOVER_LEAVE, // MoverMan need to take the mover
    DONE := 8000,     // Ablauf beendet 
    ERROR := 9000,    // Fehler 
    _max
);
END_TYPE

// ---- POUs/20_AUTO/ST105/ST105_Slider_e.TcDUT
{attribute 'qualified_only'}
{attribute 'strict'}
{attribute 'to_string'}
// slider steps for ST105 feeder
// The slider is used to separate two parts that are inside each other
TYPE ST105_Slider_e :
(
    slider_down := 0,
    slider_go_up := 10,
    slider_push_out := 20,
    slider_pusher_in := 30,
	slider_go_down := 40,
    _max
);
END_TYPE

// ---- POUs/20_AUTO/ST105/ST105_Cylinders_e.TcTLEO
{attribute 'qualified_only'}
{attribute 'strict'}
{attribute 'to_string'}
TYPE ST105_Cylinders_e :
(
    Ausschieber_ab_auf,
    Ausschieber_vor_zuruck,
    _max
);
END_TYPE

// ---- POUs/20_AUTO/ST110/ST110_Alarm_e.TcDUT
{attribute 'qualified_only'}
{attribute 'to_string'}
TYPE ST110_Alarm_e :
(
    no_error := 0,
    Axis_110_01Y_error := 1,
    Axis_110_02Z_error := 2,
    Axis_110_03Z_error := 3,
    Axis_110_04Z_error := 4,
    Cylinder_vacuum_griper_left := 5,
    Cylinder_vacuum_griper_right := 6,
    Axis_110_10W_error := 7,
    Feeder_error := 8,
    Piece_in_unused_griper := 9,
    Piece_missing_left_griper := 10,
    Piece_missing_right_griper := 11,
    Feeder_empty := 12,
    _max := 20
)BYTE;
END_TYPE

// ---- POUs/20_AUTO/ST110/ST110_Feeder_e.TcDUT
{attribute 'qualified_only'}
{attribute 'strict'}
TYPE ST110_Feeder_e :
(
    RESET := 0, // Reset

    INIT := 100, // Initialisieren 
    Init_home_table := 110,
    Init_simu_home_table := 120,
    Init_table_go_to_zero := 130,
    Init_reset_search_index := 140,
    Init_set_table_pos := 150,
    Init_see_if_piece_there := 160,

    READY := 999,  // READY to Start, Init Done 
    START := 1000, // Start Zyklisch
    check_if_feeding_necessary := 1010,
	wait_on_a_piece := 1020,
	load_piece := 1030,
	wait_rotary_table_done := 1040,

    DONE := 8000,  // Ablauf beendet 
    ERROR := 9000, // Fehler 
    _max
);
END_TYPE

// ---- POUs/20_AUTO/ST110/ST110_PnpVerPushPos_e.TcDUT
{attribute 'qualified_only'}
{attribute 'strict'}
TYPE ST110_PnpVerPushPos_e :
(
	down,
	up,
	_max
);
END_TYPE

// ---- POUs/20_AUTO/ST110/ST110_Pnp_e.TcTLEO
{attribute 'qualified_only'}
{attribute 'strict'}
{attribute 'to_string'}
TYPE
ST110_Pnp_e :
(
    RESET := 0,         // Reset
	
    INIT := 100,        // Initialisieren 
    Init_VerticalUp_04 := 110,      // move axis below the mover to its rest position
    Init_VerticalUp_02_03 := 120,   // move the axis up to rest position
	Init_HomeHorizontals := 130,
	Init_HorizontalsToTrack := 140,
	Init_stop_vacum := 150,
	Init_check_if_pces_handled := 160,
	
    MOVER_FREE_OP,      // Ab here, operation without mover can be done
    READY := 999,       // READY to Start, Init Done 
    START := 1000,      // Start Zyklisch

	PnP_Hor_ToRotTablePos := 1010,
	PnP_WaitOnFeeder := 1020,
	PnP_Ver_RotTableDown := 1030,
	Vacum_on := 1040,
	PnP_Ver_RotTableUp := 1050,
	PnP_Hor_ToTrackPos := 1060,
    waitOnMover := 1070,        // wait until the mover is there
    MOVER_NEEDED_OP,    // Since here, a mover in position is needed to perform the action

	Pnp_Handling_pin_up := 1210,
	PnP_Ver_ShuttleDown := 1220,
	PnP_Ver_StartTorqueControl := 1225, // this step is used to start the execution of the movement
	                                    // even if the torque limit is passed. This way we ensure that
										// twincat motion library accept the move_absolute command
	PnP_Ver_ShuttleTorqueControl := 1230,
	PnP_Ver_quick_stop := 1240,
	Vacum_off := 1250,
	PnP_Ver_ShuttleUp := 1260,
	
    SYNC_MOVER_LEAVE,   // MoverMan need to take the mover
    DONE := 8000,       // Ablauf beendet 
    ERROR := 9000,      // Fehler 
    _max
);
END_TYPE

// ---- POUs/20_AUTO/ST110/ST110_PnpHorPos_e.TcDUT
{attribute 'qualified_only'}
{attribute 'strict'}
TYPE ST110_PnpHorPos_e :
(
	GS,
	AS,
	_max
);
END_TYPE

// ---- POUs/20_AUTO/ST110/ST110_PnpVerPos_e.TcDUT
{attribute 'qualified_only'}
{attribute 'strict'}
TYPE ST110_PnpVerPos_e :
(
    UpEmpty,               // Up position when the Pnp is empty
    DownEmpty,             // Down position when the Pnp is picking the piece
    UpFull,                // Up position when the Pnp has gripped the piece
    DownFullQuick,         // down position with quick speed
    DownFullTorqueControl, // down position with low speed for torque control
    _max
);
END_TYPE

// ---- POUs/20_AUTO/ST110/ST110_Recipe_t.TcDUT
TYPE ST110_Recipe_t :
STRUCT
    xUseVerLeft         : BOOL; // Is the left vertical picker element is used
    xUseVerRight        : BOOL; // Is the right vertical picker element is used
    FeederConfig        : FeederDelays_t;
    waitBlowPieceTon_ms : DINT; // time to wait before to blow the piece away
    blowPieceTof_ms     : DINT; // time to let the blower take away the piece
    vakum_left_pc       : INT;  // vacum limit for left pnp
    vakum_right_pc      : INT;  // vacum limit for right pnp
END_STRUCT
END_TYPE

// ---- POUs/20_AUTO/ST115/ST115_PnpVerPushPos_e.TcDUT
{attribute 'qualified_only'}
{attribute 'strict'}
TYPE ST115_PnpVerPushPos_e :
(
	down,
	up,
	_max
);
END_TYPE

// ---- POUs/20_AUTO/ST115/ST115_Cylinders_e.TcTLEO
{attribute 'qualified_only'}
{attribute 'strict'}
{attribute 'to_string'}
TYPE ST115_Cylinders_e :
(
    GreiferLinks,
    GreiferRechts,
    _max
);
END_TYPE

// ---- POUs/20_AUTO/ST115/ST115_Recipe_t.TcDUT
TYPE ST115_Recipe_t :
STRUCT
    xUseVerLeft            : BOOL; // Is the left vertical picker element is used
    xUseVerRight           : BOOL; // Is the right vertical picker element is used
    FeederConfig           : FeederDelays_t;
END_STRUCT
END_TYPE

// ---- POUs/20_AUTO/ST115/ST115_Feeder_e.TcDUT
TYPE ST115_Feeder_e : ST110_Feeder_e;
END_TYPE

// ---- POUs/20_AUTO/ST115/ST115_PnpHorPos_e.TcDUT
TYPE ST115_PnpHorPos_e : ST110_PnpHorPos_e;
END_TYPE

// ---- POUs/20_AUTO/ST115/ST115_Pnp_e.TcTLEO
{attribute 'qualified_only'}
{attribute 'strict'}
{attribute 'to_string'}
TYPE ST115_Pnp_e :
(
    RESET := 0,         // Reset
	
    INIT := 100,        // Initialisieren 
	Init_HomeVerticals,
	Init_VerticalsUp,
	Init_HomeHorizontals,
	Init_HorizontalsToTrack,
	Init_check_if_pces_handled,
	
    MOVER_FREE_OP,      // Ab here, operation without mover can be done
    READY := 999,       // READY to Start, Init Done 
    START := 1000,      // Start Zyklisch

	PnP_Hor_ToRotTablePos,
	PnP_WaitOnFeeder,
	PnP_Ver_RotTableDown,
	Gripper_open,
	PnP_Ver_RotTableUp,
	PnP_Hor_ToTrackPos,
    waitOnMover,        // wait until the mover is there
    MOVER_NEEDED_OP,    // Since here, a mover in position is needed to perform the action

	PnP_Ver_ShuttleDown,
	PnP_Ver_ShuttleTorqueControl,
	Gripper_close,
	PnP_Ver_ShuttleUp,
	
    SYNC_MOVER_LEAVE,   // MoverMan need to take the mover
    DONE := 8000,       // Ablauf beendet 
    ERROR := 9000,      // Fehler 
    _max
);
END_TYPE

// ---- POUs/20_AUTO/ST120/ST120_Cylinders_e.TcTLEO
{attribute 'qualified_only'}
{attribute 'strict'}
{attribute 'to_string'}
TYPE ST120_Cylinders_e :
(
    GreiferLinks,
    GreiferRechts,
	SchwenkenLinks,
	SchwenkenRechts,
	HubladerLinks,
	HubladerRechts,
    _max
);
END_TYPE

// ---- POUs/20_AUTO/ST120/ST120_Feeder_e.TcDUT
{attribute 'qualified_only'}
{attribute 'strict'}
TYPE ST120_Feeder_e :
(
    RESET := 0, // Reset

    INIT := 100, // Initialisieren 
    Init_pneumatics,
	Init_pivot_to_feeder,
	Init_pivot_to_pnp,

    READY := 999,  // READY to Start, Init Done 
    START := 1000, // Start Zyklisch
    wait_tube_presence,
	wait_pnp_ready,
	rotate_to_pnp,
	wait_pce_picked,
	wait_pnp_move_out_with_the_piece,
	rotate_to_feeder,

    DONE := 8000,  // Ablauf beendet 
    ERROR := 9000, // Fehler 
    _max
);
END_TYPE

// ---- POUs/20_AUTO/ST120/ST120_PnpVerPos_e.TcDUT
TYPE ST120_PnpVerPos_e : ST110_PnpVerPos_e;
END_TYPE

// ---- POUs/20_AUTO/ST120/ST120_Pnp_e.TcTLEO
{attribute 'qualified_only'}
{attribute 'strict'}
{attribute 'to_string'}
TYPE ST120_Pnp_e :
(
    RESET := 0, // Reset

    INIT := 100, // Initialisieren 
    Init_HomeVerticals,
    Init_VerticalsUp,
    Init_HomeHorizontals,
    Init_HorizontalsToTrack,
    Init_adjust_left_clamp,
    Init_open_left_clamp,
    Init_adjust_right_clamp,
    Init_open_right_clamp,
    Init_check_if_pces_handled,

    READY := 999,  // READY to Start, Init Done 
    START := 1000, // Start Zyklisch
    MOVER_FREE_OP, // Ab here, operation without mover can be done

    PnP_Hor_ToRotTablePos,
    PnP_WaitOnFeeder,
    PnP_Ver_RotTableDown,
    Gripper_close,
    PnP_Ver_RotTableUp,
    PnP_Hor_ToTrackPos,
    waitOnMover,     // wait until the mover is there
    MOVER_NEEDED_OP, // Since here, a mover in position is needed to perform the action

    PnP_Ver_ShuttleDown,
    PnP_Ver_ShuttleTorqueControl,
    Gripper_open,
    PnP_Ver_ShuttleUp,

    SYNC_MOVER_LEAVE, // MoverMan need to take the mover
    DONE := 8000,     // Ablauf beendet 
    ERROR := 9000,    // Fehler 
    _max
);
END_TYPE

// ---- POUs/20_AUTO/ST120/ST120_Recipe_t.TcDUT
TYPE ST120_Recipe_t :
STRUCT
    xUseVerLeft               : BOOL; // Is the left vertical picker element is used
    xUseVerRight              : BOOL; // Is the right vertical picker element is used
    FeederConfigLeft          : FeederDelays_t;
    FeederConfigRight         : FeederDelays_t;
    TON_PieceInSeperatorLeft  : DINT; // TON waiting time after sensor has detected a presensce (left)
    TON_PieceInSeperatorRight : DINT; // TON waiting time after sensor has detected a presensce (right)
END_STRUCT
END_TYPE

// ---- POUs/20_AUTO/ST125/ST125_Alarm_e.TcDUT
{attribute 'qualified_only'}
{attribute 'to_string'}
TYPE ST125_Alarm_e :
(
    no_error := 0,
    Axis_120_01Y_error := 1,
    Axis_120_02Z_error := 2,
    Cylinder_griper_filterhut_left := 3,
    Cylinder_griper_filterhut_right := 4,
    Cylinder_handling_solerohr_left := 5,
    Cylinder_handling_solerohr_right := 6,
    Cylinder_griper_solerohr_left := 7,
    Cylinder_griper_solerohr_right := 8,
    Piece_in_unused_griper := 9,
    Piece_missing_left_griper := 10,
    Piece_missing_right_griper := 11,
    Feeder_empty := 12,
    Feeder_error := 13,
    Axis_120_10W_error := 14,
    Distance_sensor_dirty := 15,

    _max := 20
) BYTE;
END_TYPE

// ---- POUs/20_AUTO/ST125/ST125_Cylinders_e.TcTLEO
{attribute 'qualified_only'}
{attribute 'strict'}
{attribute 'to_string'}
TYPE ST125_Cylinders_e :
(
    GreiferFilterhutLinks,
    GreiferFilterhutRechts,
    HandlingSolerohrLinks,
    HandlingSolerohrRechts,
    GreiferSolerohrLinks,
    GreiferSolerohrRechts,
    _max
);
END_TYPE

// ---- POUs/20_AUTO/ST125/ST125_Feeder_e.TcDUT
TYPE ST125_Feeder_e : ST110_Feeder_e;
END_TYPE

// ---- POUs/20_AUTO/ST125/ST125_PnpHorPos_e.TcDUT
TYPE ST125_PnpHorPos_e : ST110_PnpHorPos_e;
END_TYPE

// ---- POUs/20_AUTO/ST125/ST125_PnpVerPos_e.TcDUT
{attribute 'qualified_only'}
{attribute 'strict'}
TYPE ST125_PnpVerPos_e :
(
    UpEmpty,               // Up position when the Pnp is empty
    DownEmpty,             // Down position when the Pnp is picking the piece
    UpFull,                // Up position when the Pnp has gripped the piece
    DownFullQuick,         // down position with quick speed
    DownFullTorqueControl, // down position with low speed for torque control
    UpToHandling,          // Go up until the handling tool can move
    _max
);
END_TYPE

// ---- POUs/20_AUTO/ST125/ST125_Pnp_e.TcTLEO
{attribute 'qualified_only'}
{attribute 'strict'}
{attribute 'to_string'}
TYPE ST125_Pnp_e :
(
    RESET := 0, // Reset

    INIT := 100, // Initialisieren 
    Init_HomeVerticals,
    Init_VerticalsUp,
	Init_open_solenohr_gripper,
	Init_handling_up,
    Init_HomeHorizontals,
    Init_HorizontalsToTrack,
    Init_adjust_left_clamp,
    Init_open_left_clamp,
    Init_adjust_right_clamp,
    Init_open_right_clamp,
    Init_check_if_pces_handled,

    MOVER_FREE_OP, // Ab here, operation without mover can be done
    READY := 999,  // READY to Start, Init Done 
    START := 1000, // Start Zyklisch

    Pnp_Hor_ToRotTablePos,
    Pnp_WaitOnFeeder,
    Pnp_Ver_RotTableDown,
    Pnp_takeTubeCap,
    Pnp_Ver_RotTableUp,
    Pnp_Hor_ToTrackPos,
    waitOnMover,     // wait until the mover is there
    MOVER_NEEDED_OP, // Since here, a mover in position is needed to perform the action

    Pnp_HandlingDown,
    Pnp_closeTubeGriper,
    Pnp_Ver_ShuttleDown,
	Pnp_Wait_on_tube_griper, // Used to catch xOUT_DONE flag from the motor
    Pnp_placeCap,
    Pnp_Ver_pushCapTorqueControl,
	PnP_Ver_quick_stop,
    Pnp_Ver_ShuttleUpToHandling,
    Pnp_HandlingSolerohrRelease,
    Pnp_Ver_ShuttleFullUp,
    Pnp_HandlingUp,

    SYNC_MOVER_LEAVE, // MoverMan need to take the mover
    DONE := 8000,     // Ablauf beendet 
    ERROR := 9000,    // Fehler 
    _max
);
END_TYPE

// ---- POUs/20_AUTO/ST125/ST125_Recipe_t.TcDUT
TYPE ST125_Recipe_t :
STRUCT
    xUseVerLeft           : BOOL; // Is the left vertical picker element is used
    xUseVerRight          : BOOL; // Is the right vertical picker element is used
    FeederConfig          : FeederDelays_t;
    diPieceGoodMaxHeight  : DINT; // Good piece maximum value (value is the output of the analog board)
    diPieceGoodMinHeight  : DINT; // Good piece minimum value (value is the output of the analog board)
    diPieceWrongMaxHeight : DINT; // Bad piece maximum value (value is the output of the analog board)
    diPieceWrongMinHeight : DINT; // Bad piece minimum value (value is the output of the analog board)
    TON_WaitPieceTime     : DINT; // additionnal waiting time of a piece to ensure the mesure is done correctly
    kraft_left_raw        : REAL; // force limit for left pnp, raw value
    kraft_right_raw       : REAL; // force limit for right pnp, raw value
END_STRUCT
END_TYPE

// ---- POUs/20_AUTO/ST128/ST128_Recipe_t.TcDUT
TYPE ST128_Recipe_t :
STRUCT
    xIsTypeMiniOrSmart    : BOOL; // do we have 2 pieces (smart and mini) or just one (others)
END_STRUCT
END_TYPE

// ---- POUs/20_AUTO/ST130/ST130_Cylinders_e.TcTLEO
TYPE ST130_Cylinders_e :
(
    Kammer_Offnen_Links,
    Kammer_Offnen_Rechts,
    Kammer_nachfullen_Links,
    Kammer_nachfullen_Rechts,
    Vibrieren_Kammer_Links,
    Vibrieren_Kammer_Rechts,
    Niederhalter_Patrone,
    Vibrienren_Patrone_Links,
    Viebrieren_Patrone_Rechts
);
END_TYPE

// ---- POUs/20_AUTO/ST130/ST130_PatroneAushebenPos_e.TcDUT
TYPE ST130_PatroneAushebenPos_e :
(
    down_GS,
    up_AS,
    _max
);
END_TYPE

// ---- POUs/20_AUTO/ST130/ST130_Recipe_t.TcDUT
TYPE ST130_Recipe_t :
STRUCT
    diLoadKammer_ms   : DINT; // waiting time until Kammer (chambre) is fully loaded
    diLoadPatrone_ms  : DINT; // waiting time until Patrone (cartridge) is fully loaded
    uiVibroUnderneath : UINT; // underneath vibro force expressed as a percentage
    xUseVerLeft       : BOOL; // Is the left vertical picker element is used
    xUseVerRight      : BOOL; // Is the right vertical picker element is used
END_STRUCT
END_TYPE

// ---- POUs/20_AUTO/ST130/ST130_Dose_e.TcTLEO
{attribute 'qualified_only'}
{attribute 'strict'}
{attribute 'to_string'}
TYPE
ST130_Dose_e :
(
    RESET := 0, // Reset

    INIT := 100, // Initialisieren 
    Init_HomeVertical_02,
    Init_Vertical_01Z_at_position,
    Init_HomeVertical_10,
    Init_Vertical_10_Down,
    Init_close_down_feeder,
    Init_close_up_feeder,
	Init_clamp_up,

    READY := 999,  // READY to Start, Init Done 
    START := 1000, // Start Zyklisch
  
    Adjust_Vertical_01Z_position, // add the offset
	open_up_feeder_first, // we ensure that the up clamp is open
	fill_kammer, // we have to wait until the kammer is full 
	
    waitOnMover,     // wait until the mover is there
    MOVER_NEEDED_OP, // Ab here, a mover in position is needed to perform the action

    check_filterhut_presence,      // when the shuttle is at position, we control the presence of the filterhut
	close_up_feeder,
    lift_up_piece_in_workposition, // we lift the piece to place it in the funel
	open_down_feeder,
    load_powder_and_vibrate,
    close_down_feeder,
    release_piece_and_open_up_feeder,
	open_up_feeder,
	clamp_down,
	clamp_up,

    SYNC_MOVER_LEAVE, // MoverMan need to take the mover
    MOVER_FREE_OP,    // here, operation without mover can be done.

    DONE := 8000,  // Ablauf beendet 
    ERROR := 9000, // Fehler 
    _max
);
END_TYPE

(*
back to shuttle
check level NIO Box
*)

// ---- POUs/20_AUTO/ST140/LaserPlace_e.TcDUT
{attribute 'qualified_only'}
{attribute 'strict'}
TYPE LaserPlace_e :
(
    NearTrack := 0,
    NearDoor := 1
);
END_TYPE

// ---- POUs/20_AUTO/ST140/ST140_Measure_e.TcTLEO
{attribute 'qualified_only'}
{attribute 'strict'}
{attribute 'to_string'}
TYPE
ST140_Measure_e :
(
    RESET := 0, // Reset

    INIT := 100, // Initialisieren 

    READY := 999,  // READY to Start, Init Done 
    START := 1000, // Start Zyklisch

    waitOnMover,     // wait until the mover is there
    MOVER_NEEDED_OP, // Ab here, a mover in position is needed to perform the action

    Measure_right,
    Move_shuttle_relative_right,
    Move_shuttle_to_pos_left,
    Measure_left,
    Move_shuttle_relative_left,
    Save_result_in_mover,

    SYNC_MOVER_LEAVE, // MoverMan need to take the mover
    MOVER_FREE_OP,    // here, operation without mover can be done.

    DONE := 8000,  // Ablauf beendet 
    ERROR := 9000, // Fehler 
    _max
);
END_TYPE

(*
back to shuttle
check level NIO Box
*)

// ---- POUs/20_AUTO/ST140/ST140_Recipe_t.TcDUT
TYPE ST140_Recipe_t :
STRUCT
    rMinHeightSensorLeft  : REAL; // minimum height allowed to be measured by the sensor
    rMaxHeightSensorLeft  : REAL; // maximum height allowed to be measured by the sensor
    rMinHeightSensorRight : REAL; // minimum height allowed to be measured by the sensor
    rMaxHeightSensorRight : REAL; // maximum height allowed to be measured by the sensor
    xIsTypeMiniOrSmart    : BOOL; // do we have 2 pieces (smart and mini) or just one (others)
END_STRUCT
END_TYPE

// ---- POUs/20_AUTO/ST145/ST145_Feeder_e.TcDUT
TYPE ST145_Feeder_e : ST110_Feeder_e;
END_TYPE

// ---- POUs/20_AUTO/ST145/ST145_PnpHorPos_e.TcDUT
TYPE ST145_PnpHorPos_e : ST110_PnpHorPos_e;
END_TYPE

// ---- POUs/20_AUTO/ST145/ST145_PnpVerPos_e.TcDUT
TYPE ST145_PnpVerPos_e : ST110_PnpVerPos_e;
END_TYPE

// ---- POUs/20_AUTO/ST145/ST145_Recipe_t.TcDUT
TYPE ST145_Recipe_t :
STRUCT
    xUseVerLeft  : BOOL; // Is the left vertical picker element is used
    xUseVerRight : BOOL; // Is the right vertical picker element is used
    FeederConfig : FeederDelays_t;
END_STRUCT
END_TYPE

// ---- POUs/20_AUTO/ST145/ST145_Pnp_e.TcTLEO
{attribute 'qualified_only'}
{attribute 'strict'}
{attribute 'to_string'}
TYPE ST145_Pnp_e :
(
    RESET := 0, // Reset

    INIT := 100, // Initialisieren 
    Init_HomeVerticals,
    Init_VerticalsUp,
    Init_HomeHorizontals,
    Init_HorizontalsToTrack,
    Init_check_if_pces_handled,

    MOVER_FREE_OP, // Ab here, operation without mover can be done
    READY := 999,  // READY to Start, Init Done 
    START := 1000, // Start Zyklisch

    PnP_Hor_ToRotTablePos,
    PnP_WaitOnFeeder,
    PnP_Ver_RotTableDown,
    Vacum_on,
    PnP_Ver_RotTableUp,
    PnP_Hor_ToTrackPos,
    waitOnMover,     // wait until the mover is there
    MOVER_NEEDED_OP, // Since here, a mover in position is needed to perform the action

    PnP_Ver_ShuttleDown,
    PnP_Ver_ShuttleTorqueControl,
    Vacum_off,
	Pnp_move_a_bit_to_feeder,
    PnP_Ver_ShuttleUp,

    SYNC_MOVER_LEAVE, // MoverMan need to take the mover
    DONE := 8000,     // Ablauf beendet 
    ERROR := 9000,    // Fehler 
    _max
);
END_TYPE

// ---- POUs/20_AUTO/ST15x/ST150_Cylinders_e.TcTLEO
{attribute 'qualified_only'}
{attribute 'strict'}
{attribute 'to_string'}
TYPE ST150_Cylinders_e : 
(
	Kraftbstutzung,
	_max
);
END_TYPE

// ---- POUs/20_AUTO/ST15x/ST150_Uss_e.TcTLEO
{attribute 'qualified_only'}
{attribute 'strict'}
{attribute 'to_string'}
TYPE ST150_Uss_e :
(
    RESET := 0, // Reset

    INIT := 100, // Initialisieren 
    Init_ResetUss_maintaining_down,

    READY := 999,  // READY to Start, Init Done 
    START := 1000, // Start Zyklisch
    MOVER_FREE_OP, // Ab here, operation without mover can be done

    waitOnMover,     // wait until the mover is there
    MOVER_NEEDED_OP, // Since here, a mover in position is needed to perform the action

    check_cap_present,     // See if the sensor sees the cap
    mover_maintening_up,   // Kraftbstützung goes up
    uss_start,             // start signal is given
    uss_working,           // we wait until the uss is finished
    mover_maintening_down, // Kraftbstützung goes down
	
	// only used for xxxx_solo process
	move_shuttle_120_mm,
	wait_shuttle_in_pos,

    SYNC_MOVER_LEAVE, // MoverMan need to take the mover
    DONE := 8000,     // Ablauf beendet 
    ERROR := 9000,    // Fehler 
    _max
);
END_TYPE

// ---- POUs/20_AUTO/ST15x/Ultrasonic_IN_bits_t.TcDUT
TYPE Ultrasonic_IN_bits_t :
STRUCT
    Bereit       : BIT; // Ready for the next
    Fehler       : BIT; // Uss in error
    US_on        : BIT; // welding is in progress (ultrsonic beam)
    NullPosition : BIT; // Uss full above
END_STRUCT
END_TYPE

// ---- POUs/20_AUTO/ST15x/Ultrasonic_OUT_bits_t.TcDUT
TYPE Ultrasonic_OUT_bits_t :
STRUCT
    Start     : BIT;
    Reset     : BIT;
    Data_Hex1 : BIT;
    Data_Hex2 : BIT;
    Data_Hex4 : BIT;
    Data_Hex8 : BIT;
END_STRUCT
END_TYPE

// ---- POUs/20_AUTO/ST16x/CETA/CETA_error_handling_t.TcDUT
TYPE CETA_error_handling_t :
STRUCT
    command_in_error : CETA_IN_u;
    error_code       : BYTE;
END_STRUCT
END_TYPE

// ---- POUs/20_AUTO/ST16x/CETA/CETA_IN_bits_t.TcDUT
TYPE CETA_IN_bits_t :
STRUCT
    b08_error_bit                    : BIT; // error bit
    b09_communication_possible       : BIT; // communication possible
    b10_device_ready_to_start        : BIT; // device ready to start
    b11_result_block_handshake_bit   : BIT; // result block handshake bit
    b12_measuring_curve              : BIT; // measuring curve
    b13_res_b13                      : BIT;
    b14_res_b14                      : BIT;
    b15_res_b15                      : BIT;
    b00_measurement_complete         : BIT; // measurement complete
    b01_parameters_received          : BIT; // parameters received
    b02_parameters_available         : BIT; // parameters available
    b03_error_code_available         : BIT; // error code available
    b04_front_panel_lock_state       : BIT; // front panel lock state
    b05_program_number_assigned      : BIT; // program number assigned
    b06_system_information_available : BIT; // system information available
    b07_cycle_counter_available      : BIT; // cycle counter available
END_STRUCT
END_TYPE

// ---- POUs/20_AUTO/ST16x/CETA/CETA_IN_u.TcDUT
TYPE CETA_IN_u :
UNION
    bits : CETA_IN_bits_t;
    raw  : UINT;
END_UNION
END_TYPE

// ---- POUs/20_AUTO/ST16x/CETA/CETA_Measurement_t/CETA_Measurement_block2_t.TcDUT
{attribute 'pack_mode' := '1'}
TYPE CETA_Measurement_block2_t :
STRUCT
    Program_number       : USINT;
    Result_chanel_1      : USINT;
    Test_mode            : USINT;
    Result_chanel_2      : USINT;
    Cons_Num_Res_Block   : USINT;
    Num_Following_Blocks : USINT;
    Reserve              : USINT;
    Time_hour            : USINT;
    Time_minute          : USINT;
    Time_second          : USINT;
    Data_offset_12       : CETA_Res_Data_t;
    Data_offset_16       : CETA_Res_Data_t;
    Data_offset_20       : CETA_Res_Data_t;
    Data_offset_24       : CETA_Res_Data_t;
    Data_offset_28       : CETA_Res_Data_t;
    Data_offset_32       : CETA_Res_Data_t;
    Data_offset_36       : CETA_Res_Data_t;
    Data_offset_40       : CETA_Res_Data_t;
    Data_offset_44       : CETA_Res_Data_t;
END_STRUCT
END_TYPE

// ---- POUs/20_AUTO/ST16x/CETA/CETA_Measurement_t/CETA_Measurement_t.TcDUT
{attribute 'qualified_only'}
{attribute 'strict'}
TYPE CETA_Measurement_t :
STRUCT
	Block0 : CETA_Measurement_block1_t;
	Block1 : CETA_Measurement_block2_t;
	Block2 : CETA_Measurement_block3_t;
END_STRUCT
END_TYPE

// ---- POUs/20_AUTO/ST16x/CETA/CETA_Measurement_t/CETA_Res_Data_t.TcDUT
{attribute 'pack_mode' := '1'}
TYPE CETA_Res_Data_t :
STRUCT
    Data  : INT;
    Unit  : CETA_Unit_e;
    Digit : USINT;
END_STRUCT
END_TYPE

// ---- POUs/20_AUTO/ST16x/CETA/CETA_OUT_bits_t.TcDUT
TYPE CETA_OUT_bits_t :
STRUCT
    b08_reset_error_bit               : BIT; // reset error bit
    b09_res_b9                        : BIT; // res_b9
    b10_res_b10                       : BIT; // res_b10
    b11_request_next_result_block     : BIT; // request next result block
    b12_res_b12                       : BIT; // res_b12
    b13_res_b13                       : BIT; // res_b13
    b14_res_b14                       : BIT; // res_b14
    b15_res_b15                       : BIT; // res_b15
    b00_start_stop                    : BIT; // start / stop (stop resets the device)
    b01_send_parameters               : BIT; // send parameters
    b02_request_parameters            : BIT; // request parameters
    b03_request_error_code            : BIT; // request error code
    b04_change_front_panel_lock_state : BIT; // change front panel lock state
    b05_assign_program_number         : BIT; // assign program number
    b06_request_system_information    : BIT; // request system information
    b07_request_cycle_counter         : BIT; // request cycle counter
END_STRUCT
END_TYPE

// ---- POUs/20_AUTO/ST16x/CETA/CETA_OUT_u.TcDUT
TYPE CETA_OUT_u :
UNION
    bits : CETA_OUT_bits_t;
    raw  : UINT;
END_UNION
END_TYPE

// ---- POUs/20_AUTO/ST16x/CETA/CETA_Parameter_blocks/CETA_Parameter_blocks_t.TcDUT
TYPE CETA_Parameter_blocks_t :
STRUCT
    _00_program_name                : ARRAY[0..16] OF BYTE;
    _01_test_mode                   : ARRAY[0..27] OF BYTE;
    _02_delay                       : ARRAY[0..27] OF BYTE;
    _03_fill                        : ARRAY[0..27] OF BYTE;
    _04_stabilisation               : ARRAY[0..27] OF BYTE;
    _05_test                        : ARRAY[0..27] OF BYTE;
    _06_vent                        : ARRAY[0..27] OF BYTE;
    _07_prefill_prevent             : ARRAY[0..27] OF BYTE;
    _08_flood_sealed_component      : ARRAY[0..27] OF BYTE;
    _09_flood_sealed_high_res       : ARRAY[0..27] OF BYTE;
    _0A_fill_primary_pressure       : ARRAY[0..27] OF BYTE;
    _0B_fill_ram_pressure           : ARRAY[0..27] OF BYTE;
    _0C_automatic_function_check    : ARRAY[0..27] OF BYTE;
    _0D_temperature_compensation    : ARRAY[0..27] OF BYTE;
    _0E_control_valves              : ARRAY[0..27] OF BYTE;
    _0F_option_switch               : ARRAY[0..27] OF BYTE;
    _10_fill_reservoir              : ARRAY[0..27] OF BYTE;
    _11_correction_factor           : ARRAY[0..27] OF BYTE;
    _12_smotth_turbo_filling        : ARRAY[0..27] OF BYTE;
    _13_pressure_stages             : ARRAY[0..27] OF BYTE;
    _14_test_channel_two            : ARRAY[0..27] OF BYTE;
    _15_usb_measurement_curve_id    : ARRAY[0..27] OF BYTE;
    _16_program_series              : ARRAY[0..27] OF BYTE;
    _17_primary_prefill_pressure    : ARRAY[0..27] OF BYTE;
    _18_primary_pressure_smooth     : ARRAY[0..27] OF BYTE;
    _19_nc                          : ARRAY[0..27] OF BYTE;
    _1A_test_repetition             : ARRAY[0..27] OF BYTE;
    _1B_test_repetition_channel_two : ARRAY[0..27] OF BYTE;
    _1C_exponential_extrapolation   : ARRAY[0..27] OF BYTE;
    _1D_pulse                       : ARRAY[0..27] OF BYTE;
    _1E_vent_to                     : ARRAY[0..27] OF BYTE;
    _1F_reference_atmosphere        : ARRAY[0..27] OF BYTE;
END_STRUCT
END_TYPE

// ---- POUs/20_AUTO/ST16x/CETA/CETA_com_union/CETA_Parameter_blocks_u.TcDUT
TYPE CETA_Parameter_blocks_u :
UNION
	as_struct : CETA_Parameter_blocks_t;
	as_2d_array : ARRAY[0..16#1F] OF ARRAY[0..59] OF BYTE;
END_UNION
END_TYPE

// ---- POUs/20_AUTO/ST16x/CETA/CETA_Result_e.TcDUT
{attribute 'qualified_only'}
{attribute 'strict'}
TYPE CETA_Result_e :
(
	OK := 1,
	NOK := 2
)USINT;
END_TYPE

// ---- POUs/20_AUTO/ST16x/CETA/CETA_Unit_e.TcDUT
{attribute 'qualified_only'}
{attribute 'strict'}
{attribute 'to_string'}
TYPE CETA_Unit_e :
(
    Pa := 000,
    Pa_per_s := 001,
    ml_per_min := 002,
    ml_per_h := 003,
    mbar := 004,
    bar := 005,
    ml_per_min_2 := 006,
    mbar_times_l_per_s := 007,
    l_per_h := 008,
    hPa_per_s := 009,
    PSI := 010,
    PSI_per_s := 011,
    hPa := 012,
    l_per_min := 013,
    ml_per_h_2 := 014,
    s_ := 017,
    percent := 018,
    mbar_per_s := 019,
    bar_per_s := 020,
    ms := 021,
    mmHg := 022,
    mmWs := 023,
    Torr := 024,
    V := 214,
    deg_C := 215,
    cm_3 := 216,
    ml := 217,
    _no_unit := 218,
    L := 219,
    deg_F := 220,
    _no_unit_254 := 254,
    _no_unit_255 := 255
)USINT;
END_TYPE

// ---- POUs/20_AUTO/ST16x/ST160_PnpVerPos_e.TcDUT
{attribute 'qualified_only'}
{attribute 'to_string'}
TYPE ST160_PnpVerPos_e:
(
	gs_down,
	as_up,
	_max
);
END_TYPE

// ---- POUs/20_AUTO/ST16x/ST160_Cylinders_e.TcTLEO
{attribute 'qualified_only'}
{attribute 'strict'}
{attribute 'to_string'}
TYPE ST160_Cylinders_e : 
(
	Niederhalter_links,
	Niederhalter_rechts,
	Dichtung_prufglocke_links,
	Dichtung_prufglocke_rechts,
	nc_160_06,
	nc_160_07,
	_max
);
END_TYPE

// ---- POUs/20_AUTO/ST16x/ST160_Recipe_t.TcDUT
TYPE ST160_Recipe_t :
STRUCT
    Use_element_left : BOOL; //a 
    Use_element_right : BOOL; // 
END_STRUCT
END_TYPE

// ---- POUs/20_AUTO/ST16x/ST160_CETA_e.TcTLEO
{attribute 'qualified_only'}
{attribute 'strict'}
{attribute 'to_string'}
TYPE ST160_CETA_e :
(
    RESET := 0, // Reset

    INIT := 100, // Initialisieren 
    Init_pneumatics,
    Init_vertical_down,
    Init_set_program_number,

    READY := 999,  // READY to Start, Init Done 
    START := 1000, // Start Zyklisch

    waitOnMover,     // wait until the mover is there
    MOVER_NEEDED_OP, // Since here, a mover in position is needed to perform the action

    handling_down,       // 
    vertical_up,   // 
    seal_piece,          //
    CETA_start,    // 
    CETA_wait_on_result, // 
    CETA_read,     // 
    unseal_piece,        //
    vertical_down, // 
    handling_up,         // 

    SYNC_MOVER_LEAVE, // MoverMan need to take the mover
    MOVER_FREE_OP,       // Ab here, operation without mover can be done

    DONE := 8000,  // Ablauf beendet 
    ERROR := 9000, // Fehler 
    _max
);
END_TYPE

// ---- POUs/20_AUTO/ST170/ST170_RFID_e.TcTLEO
{attribute 'qualified_only'}
{attribute 'strict'}
{attribute 'to_string'}
TYPE ST170_RFID_e :
(
    RESET := 0, // Reset

    INIT := 100, // Initialisieren 
    Init_vertical_homing,
    Init_vertical_down,

    READY := 999,  // READY to Start, Init Done 
    START := 1000, // Start Zyklisch

    waitOnMover,     // wait until the mover is there
    MOVER_NEEDED_OP, // Since here, a mover in position is needed to perform the action

    vertical_up,         // 
    RFID_start,    // 
    RFID_wait_on_result, // 
    RFID_read,     // 
    vertical_down,       // 

    SYNC_MOVER_LEAVE, // MoverMan need to take the mover
    MOVER_FREE_OP,       // Ab here, operation without mover can be done

    DONE := 8000,  // Ablauf beendet 
    ERROR := 9000, // Fehler 
    _max
);
END_TYPE

// ---- POUs/20_AUTO/ST170/ST170_PnpVerPos_e.TcDUT
{attribute 'qualified_only'}
{attribute 'to_string'}
TYPE ST170_PnpVerPos_e:
(
	gs_down,
	as_up,
	_max
);
END_TYPE

// ---- POUs/20_AUTO/ST170/ST170_Recipe_t.TcDUT
TYPE ST170_Recipe_t :
STRUCT
    Use_element_left  : BOOL; //a 
    Use_element_right : BOOL; // 
	RFID_Type         : USINT; 
END_STRUCT
END_TYPE

// ---- POUs/20_AUTO/ST175/ST175_LASER_e.TcTLEO
{attribute 'qualified_only'}
{attribute 'strict'}
{attribute 'to_string'}
TYPE ST175_LASER_e :
(
    RESET := 0, // Reset

    INIT := 100, // Initialisieren 
    Init_pneumatics := 110,
	Init_laser_warmup := 120,

    READY := 999,  // READY to Start, Init Done 
    START := 1000, // Start Zyklisch
    MOVER_FREE_OP, // Ab here, operation without mover can be done

    waitOnMover,     // wait until the mover is there
    MOVER_NEEDED_OP, // Since here, a mover in position is needed to perform the action

    close_doors := 1100, // 
    handling_down := 1110,          // 
    LASER_start := 1120, // 
    LASER_wait_on_finish := 1130, // 
    handling_up := 1140, // 
	move_shuttle_to_left_piece := 1150,
	wait_shuttle_in_place := 1160,
    open_doors := 1170, // 

    SYNC_MOVER_LEAVE, // MoverMan need to take the mover
    DONE := 8000,     // Ablauf beendet 
    ERROR := 9000,    // Fehler 
    _max
);
END_TYPE

// ---- POUs/20_AUTO/ST175/ST175_Cylinders_e.TcTLEO
{attribute 'qualified_only'}
{attribute 'strict'}
{attribute 'to_string'}
TYPE ST175_Cylinders_e : 
(
	Niederhalter,
	Door_entry,
	Door_exit,
	_max
);
END_TYPE

// ---- POUs/20_AUTO/ST175/ST175_Recipe_t.TcDUT
TYPE ST175_Recipe_t :
STRUCT
    isTypeSmartOrMini : BOOL; // do we need to run the laser twice on the same mover?
    file_name         : STRING;
END_STRUCT
END_TYPE

// ---- POUs/20_AUTO/ST175/Trumpf/if_Command_t.TcDUT
{attribute 'pack_mode' := '1'}
TYPE if_Command_t :
STRUCT
    iTlvHandshake : INT;
    diTlvTag      : DINT;
    diTlvLenght   : DINT;
    abyTlvValues  : ARRAY[0..117] OF BYTE;
    bit_command   : if_BitCommand_u;
END_STRUCT
END_TYPE

// ---- POUs/20_AUTO/ST175/Trumpf/if_Command_u.TcDUT
TYPE if_Command_u :
UNION
    as_word_array : ARRAY[0..63] OF WORD;
    as_struct     : if_Command_t;
END_UNION
END_TYPE

// ---- POUs/20_AUTO/ST180/ST180_Cylinders_e.TcTLEO
TYPE ST180_Cylinders_e :
(
    Greifer_Patrone_Links,
    Greifer_Patrone_Rechts,
    Niederhalter_Deckel_Links,
    Niederhalter_Deckel_Rechts
);
END_TYPE

// ---- POUs/20_AUTO/ST180/ST180_PnpVerPos_e.TcDUT
TYPE ST180_PnpVerPos_e :
(
    up_empty,
    down_empty,
    up_full,
    down_full,
    _max
);
END_TYPE

// ---- POUs/20_AUTO/ST180/ST180_Pnp_e.TcTLEO
{attribute 'qualified_only'}
{attribute 'strict'}
{attribute 'to_string'}
TYPE
ST180_Pnp_e :
(
    RESET := 0, // Reset

